LIN {X 0,Y 513.957,Z 334.017,A -85,B 0,C 180,E1 -12997.827,E2 -12997.827} C_VEL
LIN {X 0,Y 513.921,Z 334.019,A -85,B 0,C 180,E1 -13000.86,E2 -13000.86} C_VEL
LIN {X 0,Y 513.953,Z 334.017,A -85,B 0,C 180,E1 -13003.754,E2 -13003.754} C_VEL
LIN {X 0,Y 513.947,Z 334.027,A -85,B 0,C 180,E1 -13007.044,E2 -13007.044} C_VEL
LIN {X 0,Y 513.919,Z 334.024,A -85,B 0,C 180,E1 -13010.164,E2 -13010.164} C_VEL
LIN {X 0,Y 513.918,Z 334.026,A -85,B 0,C 180,E1 -13013.527,E2 -13013.527} C_VEL
LIN {X 0,Y 513.913,Z 334.024,A -85,B 0,C 180,E1 -13016.243,E2 -13016.243} C_VEL
LIN {X 0,Y 513.986,Z 334.221,A -85,B 0,C 180,E1 -13019.321,E2 -13019.321} C_VEL
LIN {X 0,Y 517.909,Z 351.016,A -85,B 0,C 180,E1 -13021.747,E2 -13021.747} C_VEL
LIN {X 0,Y 519.515,Z 360.152,A -85,B 0,C 180,E1 -13023.008,E2 -13023.008} C_VEL
LIN {X 0,Y 518.072,Z 381.283,A -85,B 0,C 180,E1 -13025.646,E2 -13025.646} C_VEL
LIN {X 0,Y 516.469,Z 407.915,A -85,B 0,C 180,E1 -13028.937,E2 -13028.937} C_VEL
LIN {X 0,Y 515.682,Z 421.479,A -85,B 0,C 180,E1 -13030.575,E2 -13030.575} C_VEL
LIN {X 0,Y 517.921,Z 437.713,A -85,B 0,C 180,E1 -13031.06,E2 -13031.06} C_VEL
LIN {X 0,Y 519.767,Z 455.53,A -85,B 0,C 180,E1 -13031.51,E2 -13031.51} C_VEL
LIN {X 0,Y 521.044,Z 469.937,A -85,B 0,C 180,E1 -13031.766,E2 -13031.766} C_VEL
LIN {X 0,Y 519.855,Z 563.729,A -85,B 0,C 180,E1 -13033.083,E2 -13033.083} C_VEL
LIN {X 0,Y 519.209,Z 578.333,A -85,B 0,C 180,E1 -13033.441,E2 -13033.441} C_VEL
LIN {X 0,Y 518.369,Z 591.708,A -85,B 0,C 180,E1 -13033.918,E2 -13033.918} C_VEL
LIN {X 0,Y 517.524,Z 603.945,A -85,B 0,C 180,E1 -13034.496,E2 -13034.496} C_VEL
LIN {X 0,Y 516.53,Z 616.831,A -85,B 0,C 180,E1 -13035.27,E2 -13035.27} C_VEL
LIN {X 0,Y 515.468,Z 629.745,A -85,B 0,C 180,E1 -13036.243,E2 -13036.243} C_VEL
LIN {X 0,Y 514.622,Z 640.615,A -85,B 0,C 180,E1 -13037.222,E2 -13037.222} C_VEL
LIN {X 0,Y 514.134,Z 652.534,A -85,B 0,C 180,E1 -13038.208,E2 -13038.208} C_VEL
LIN {X 0,Y 513.612,Z 663.514,A -85,B 0,C 180,E1 -13039.313,E2 -13039.313} C_VEL
LIN {X 0,Y 513.218,Z 673.738,A -85,B 0,C 180,E1 -13040.574,E2 -13040.574} C_VEL
LIN {X 0,Y 512.862,Z 681.617,A -85,B 0,C 180,E1 -13041.755,E2 -13041.755} C_VEL
LIN {X 0,Y 512.651,Z 688.156,A -85,B 0,C 180,E1 -13042.936,E2 -13042.936} C_VEL
LIN {X 0,Y 512.551,Z 693.504,A -85,B 0,C 180,E1 -13044.117,E2 -13044.117} C_VEL
LIN {X 0,Y 512.438,Z 697.792,A -85,B 0,C 180,E1 -13045.296,E2 -13045.296} C_VEL
LIN {X 0,Y 512.414,Z 700.648,A -85,B 0,C 180,E1 -13046.264,E2 -13046.264} C_VEL
LIN {X 0,Y 512.391,Z 703.639,A -85,B 0,C 180,E1 -13047.649,E2 -13047.649} C_VEL
LIN {X 0,Y 512.384,Z 705.592,A -85,B 0,C 180,E1 -13049.217,E2 -13049.217} C_VEL
LIN {X 0,Y 512.384,Z 706.077,A -85,B 0,C 180,E1 -13050.783,E2 -13050.783} C_VEL
LIN {X 0,Y 512.395,Z 705.11,A -85,B 0,C 180,E1 -13052.35,E2 -13052.35} C_VEL
LIN {X 0,Y 512.438,Z 702.692,A -85,B 0,C 180,E1 -13053.919,E2 -13053.919} C_VEL
LIN {X 0,Y 512.588,Z 698.767,A -85,B 0,C 180,E1 -13055.489,E2 -13055.489} C_VEL
LIN {X 0,Y 512.786,Z 694.711,A -85,B 0,C 180,E1 -13056.667,E2 -13056.667} C_VEL
LIN {X 0,Y 513.044,Z 689.687,A -85,B 0,C 180,E1 -13057.847,E2 -13057.847} C_VEL
LIN {X 0,Y 513.489,Z 682.439,A -85,B 0,C 180,E1 -13059.223,E2 -13059.223} C_VEL
LIN {X 0,Y 514.068,Z 674.823,A -85,B 0,C 180,E1 -13060.401,E2 -13060.401} C_VEL
LIN {X 0,Y 514.707,Z 665.365,A -85,B 0,C 180,E1 -13061.615,E2 -13061.615} C_VEL
LIN {X 0,Y 515.541,Z 654.607,A -85,B 0,C 180,E1 -13062.755,E2 -13062.755} C_VEL
LIN {X 0,Y 516.298,Z 643.373,A -85,B 0,C 180,E1 -13063.734,E2 -13063.734} C_VEL
LIN {X 0,Y 517.195,Z 631.022,A -85,B 0,C 180,E1 -13064.61,E2 -13064.61} C_VEL
LIN {X 0,Y 518.024,Z 617.389,A -85,B 0,C 180,E1 -13065.388,E2 -13065.388} C_VEL
LIN {X 0,Y 518.795,Z 603.147,A -85,B 0,C 180,E1 -13066.018,E2 -13066.018} C_VEL
LIN {X 0,Y 519.42,Z 589.095,A -85,B 0,C 180,E1 -13066.469,E2 -13066.469} C_VEL
LIN {X 0,Y 520.013,Z 571.059,A -85,B 0,C 180,E1 -13066.846,E2 -13066.846} C_VEL
LIN {X 0,Y 522.738,Z 481.781,A -85,B 0,C 180,E1 -13068.556,E2 -13068.556} C_VEL
LIN {X 0,Y 523.003,Z 467.316,A -85,B 0,C 180,E1 -13068.858,E2 -13068.858} C_VEL
LIN {X 0,Y 521.545,Z 448.408,A -85,B 0,C 180,E1 -13069.366,E2 -13069.366} C_VEL
LIN {X 0,Y 519.936,Z 435.629,A -85,B 0,C 180,E1 -13069.758,E2 -13069.758} C_VEL
LIN {X 0,Y 517.568,Z 410.308,A -85,B 0,C 180,E1 -13070.964,E2 -13070.964} C_VEL
LIN {X 0,Y 516.066,Z 396.877,A -85,B 0,C 180,E1 -13071.707,E2 -13071.707} C_VEL
LIN {X 0,Y 517.095,Z 376.419,A -85,B 0,C 180,E1 -13074.19,E2 -13074.19} C_VEL
LIN {X 0,Y 518.269,Z 355.713,A -85,B 0,C 180,E1 -13076.72,E2 -13076.72} C_VEL
LIN {X 0,Y 515.192,Z 339.734,A -85,B 0,C 180,E1 -13078.859,E2 -13078.859} C_VEL
LIN {X 0,Y 514.001,Z 334.02,A -85,B 0,C 180,E1 -13079.659,E2 -13079.659} C_VEL
LIN {X 0,Y 513.908,Z 334.025,A -85,B 0,C 180,E1 -13082.323,E2 -13082.323} C_VEL
LIN {X 0,Y 513.9,Z 334.031,A -85,B 0,C 180,E1 -13085.135,E2 -13085.135} C_VEL
LIN {X 0,Y 513.895,Z 334.026,A -85,B 0,C 180,E1 -13087.832,E2 -13087.832} C_VEL
LIN {X 0,Y 513.915,Z 334.027,A -85,B 0,C 180,E1 -13090.861,E2 -13090.861} C_VEL
LIN {X 0,Y 513.942,Z 334.025,A -85,B 0,C 180,E1 -13094.033,E2 -13094.033} C_VEL
LIN {X 0,Y 513.919,Z 334.025,A -85,B 0,C 180,E1 -13097.041,E2 -13097.041} C_VEL
LIN {X 0,Y 513.918,Z 334.026,A -85,B 0,C 180,E1 -13100.165,E2 -13100.165} C_VEL
LIN {X 0,Y 513.952,Z 334.023,A -85,B 0,C 180,E1 -13103.155,E2 -13103.155} C_VEL
LIN {X 0,Y 513.933,Z 334.027,A -85,B 0,C 180,E1 -13106.24,E2 -13106.24} C_VEL
LIN {X 0,Y 513.966,Z 334.145,A -85,B 0,C 180,E1 -13106.734,E2 -13106.734} C_VEL
LIN {X 0,Y 518.504,Z 346.552,A -85,B 0,C 180,E1 -13108.863,E2 -13108.863} C_VEL
LIN {X 0,Y 522.071,Z 358.438,A -85,B 0,C 180,E1 -13110.702,E2 -13110.702} C_VEL
LIN {X 0,Y 524.202,Z 368.507,A -85,B 0,C 180,E1 -13112.117,E2 -13112.117} C_VEL
LIN {X 0,Y 522.434,Z 393.697,A -85,B 0,C 180,E1 -13115.018,E2 -13115.018} C_VEL
LIN {X 0,Y 520.704,Z 420.277,A -85,B 0,C 180,E1 -13118.029,E2 -13118.029} C_VEL
LIN {X 0,Y 519.609,Z 439.597,A -85,B 0,C 180,E1 -13120.219,E2 -13120.219} C_VEL
LIN {X 0,Y 522.629,Z 456.777,A -85,B 0,C 180,E1 -13120.791,E2 -13120.791} C_VEL
LIN {X 0,Y 523.743,Z 466.69,A -85,B 0,C 180,E1 -13121.071,E2 -13121.071} C_VEL
LIN {X 0,Y 520.924,Z 555.644,A -85,B 0,C 180,E1 -13122.771,E2 -13122.771} C_VEL
LIN {X 0,Y 520.115,Z 582.822,A -85,B 0,C 180,E1 -13123.298,E2 -13123.298} C_VEL
LIN {X 0,Y 519.488,Z 596.312,A -85,B 0,C 180,E1 -13123.703,E2 -13123.703} C_VEL
LIN {X 0,Y 518.707,Z 610.395,A -85,B 0,C 180,E1 -13124.281,E2 -13124.281} C_VEL
LIN {X 0,Y 517.916,Z 624.002,A -85,B 0,C 180,E1 -13125.01,E2 -13125.01} C_VEL
LIN {X 0,Y 517.038,Z 635.75,A -85,B 0,C 180,E1 -13125.786,E2 -13125.786} C_VEL
LIN {X 0,Y 516.1,Z 647.833,A -85,B 0,C 180,E1 -13126.76,E2 -13126.76} C_VEL
LIN {X 0,Y 515.268,Z 658.722,A -85,B 0,C 180,E1 -13127.837,E2 -13127.837} C_VEL
LIN {X 0,Y 514.613,Z 668.576,A -85,B 0,C 180,E1 -13129.015,E2 -13129.015} C_VEL
LIN {X 0,Y 513.925,Z 676.801,A -85,B 0,C 180,E1 -13130.191,E2 -13130.191} C_VEL
LIN {X 0,Y 513.376,Z 684.669,A -85,B 0,C 180,E1 -13131.566,E2 -13131.566} C_VEL
LIN {X 0,Y 512.916,Z 690.978,A -85,B 0,C 180,E1 -13132.94,E2 -13132.94} C_VEL
LIN {X 0,Y 512.627,Z 695.283,A -85,B 0,C 180,E1 -13134.118,E2 -13134.118} C_VEL
LIN {X 0,Y 512.466,Z 698.685,A -85,B 0,C 180,E1 -13135.296,E2 -13135.296} C_VEL
LIN {X 0,Y 512.357,Z 701.825,A -85,B 0,C 180,E1 -13136.865,E2 -13136.865} C_VEL
LIN {X 0,Y 512.309,Z 703.515,A -85,B 0,C 180,E1 -13138.433,E2 -13138.433} C_VEL
LIN {X 0,Y 512.306,Z 703.777,A -85,B 0,C 180,E1 -13140,E2 -13140} C_VEL
LIN {X 0,Y 512.307,Z 702.606,A -85,B 0,C 180,E1 -13141.567,E2 -13141.567} C_VEL
LIN {X 0,Y 512.328,Z 699.97,A -85,B 0,C 180,E1 -13143.135,E2 -13143.135} C_VEL
LIN {X 0,Y 512.418,Z 695.775,A -85,B 0,C 180,E1 -13144.705,E2 -13144.705} C_VEL
LIN {X 0,Y 512.523,Z 691.231,A -85,B 0,C 180,E1 -13145.968,E2 -13145.968} C_VEL
LIN {X 0,Y 512.769,Z 684.336,A -85,B 0,C 180,E1 -13147.457,E2 -13147.457} C_VEL
LIN {X 0,Y 513.092,Z 676.309,A -85,B 0,C 180,E1 -13148.835,E2 -13148.835} C_VEL
LIN {X 0,Y 513.475,Z 667.895,A -85,B 0,C 180,E1 -13150.016,E2 -13150.016} C_VEL
LIN {X 0,Y 514.049,Z 657.233,A -85,B 0,C 180,E1 -13151.251,E2 -13151.251} C_VEL
LIN {X 0,Y 514.52,Z 646.405,A -85,B 0,C 180,E1 -13152.282,E2 -13152.282} C_VEL
LIN {X 0,Y 515.135,Z 633.805,A -85,B 0,C 180,E1 -13153.265,E2 -13153.265} C_VEL
LIN {X 0,Y 515.76,Z 621.419,A -85,B 0,C 180,E1 -13154.05,E2 -13154.05} C_VEL
LIN {X 0,Y 516.376,Z 607.834,A -85,B 0,C 180,E1 -13154.735,E2 -13154.735} C_VEL
LIN {X 0,Y 516.783,Z 593.624,A -85,B 0,C 180,E1 -13155.275,E2 -13155.275} C_VEL
LIN {X 0,Y 517.198,Z 578.976,A -85,B 0,C 180,E1 -13155.665,E2 -13155.665} C_VEL
LIN {X 0,Y 519.097,Z 462.644,A -85,B 0,C 180,E1 -13157.655,E2 -13157.655} C_VEL
LIN {X 0,Y 516.428,Z 439.504,A -85,B 0,C 180,E1 -13158.152,E2 -13158.152} C_VEL
LIN {X 0,Y 517.63,Z 410.077,A -85,B 0,C 180,E1 -13161.43,E2 -13161.43} C_VEL
LIN {X 0,Y 518.796,Z 384.213,A -85,B 0,C 180,E1 -13164.318,E2 -13164.318} C_VEL
LIN {X 0,Y 519.838,Z 360.3,A -85,B 0,C 180,E1 -13167.003,E2 -13167.003} C_VEL
LIN {X 0,Y 515.28,Z 339.725,A -85,B 0,C 180,E1 -13169.543,E2 -13169.543} C_VEL
LIN {X 0,Y 514.013,Z 334.014,A -85,B 0,C 180,E1 -13170.278,E2 -13170.278} C_VEL
LIN {X 0,Y 513.973,Z 334.022,A -85,B 0,C 180,E1 -13173.033,E2 -13173.033} C_VEL
LIN {X 0,Y 513.984,Z 334.015,A -85,B 0,C 180,E1 -13175.874,E2 -13175.874} C_VEL
LIN {X 0,Y 513.947,Z 334.025,A -85,B 0,C 180,E1 -13179.028,E2 -13179.028} C_VEL
LIN {X 0,Y 513.958,Z 334.017,A -85,B 0,C 180,E1 -13181.897,E2 -13181.897} C_VEL
LIN {X 0,Y 513.974,Z 334.021,A -85,B 0,C 180,E1 -13185.126,E2 -13185.126} C_VEL
LIN {X 0,Y 513.959,Z 334.018,A -85,B 0,C 180,E1 -13188.103,E2 -13188.103} C_VEL
LIN {X 0,Y 513.952,Z 334.023,A -85,B 0,C 180,E1 -13190.972,E2 -13190.972} C_VEL
LIN {X 0,Y 513.984,Z 334.016,A -85,B 0,C 180,E1 -13194.127,E2 -13194.127} C_VEL
LIN {X 0,Y 513.962,Z 334.02,A -85,B 0,C 180,E1 -13196.966,E2 -13196.966} C_VEL
LIN {X 0,Y 513.952,Z 334.019,A -85,B 0,C 180,E1 -13199.718,E2 -13199.718} C_VEL
LIN {X 0,Y 513.973,Z 334.024,A -85,B 0,C 180,E1 -13202.396,E2 -13202.396} C_VEL
LIN {X 0,Y 513.933,Z 334.022,A -85,B 0,C 180,E1 -13205.007,E2 -13205.007} C_VEL
LIN {X 0,Y 513.995,Z 334.017,A -85,B 0,C 180,E1 -13207.922,E2 -13207.922} C_VEL
LIN {X 0,Y 513.97,Z 334.017,A -85,B 0,C 180,E1 -13210.909,E2 -13210.909} C_VEL
LIN {X 0,Y 513.973,Z 334.017,A -85,B 0,C 180,E1 -13213.37,E2 -13213.37} C_VEL
LIN {X 0,Y 514.062,Z 334.012,A -85,B 0,C 180,E1 -13215.803,E2 -13215.803} C_VEL
LIN {X 0,Y 514.031,Z 334.01,A -85,B 0,C 180,E1 -13216.922,E2 -13216.922} C_VEL
LIN {X 0,Y 519.318,Z 349.174,A -85,B 0,C 180,E1 -13217.334,E2 -13217.334} C_VEL
LIN {X 0,Y 520.205,Z 352.303,A -85,B 0,C 180,E1 -13217.408,E2 -13217.408} C_VEL
LIN {X 0,Y 519.393,Z 423.895,A -85,B 0,C 180,E1 -13218.392,E2 -13218.392} C_VEL
LIN {X 0,Y 518.705,Z 429.739,A -85,B 0,C 180,E1 -13218.451,E2 -13218.451} C_VEL
LIN {X 0,Y 513.062,Z 448.73,A -85,B 0,C 180,E1 -13218.548,E2 -13218.548} C_VEL
LIN {X 0,Y 512.399,Z 454.555,A -85,B 0,C 180,E1 -13218.625,E2 -13218.625} C_VEL
LIN {X 0,Y 512.285,Z 468.637,A -85,B 0,C 180,E1 -13218.964,E2 -13218.964} C_VEL
LIN {X 0,Y 512.007,Z 482.396,A -85,B 0,C 180,E1 -13219.457,E2 -13219.457} C_VEL
LIN {X 0,Y 511.557,Z 494.768,A -85,B 0,C 180,E1 -13220.046,E2 -13220.046} C_VEL
LIN {X 0,Y 511.014,Z 507.231,A -85,B 0,C 180,E1 -13220.802,E2 -13220.802} C_VEL
LIN {X 0,Y 510.442,Z 519.295,A -85,B 0,C 180,E1 -13221.716,E2 -13221.716} C_VEL
LIN {X 0,Y 509.72,Z 529.971,A -85,B 0,C 180,E1 -13222.697,E2 -13222.697} C_VEL
LIN {X 0,Y 508.908,Z 540.524,A -85,B 0,C 180,E1 -13223.877,E2 -13223.877} C_VEL
LIN {X 0,Y 508.264,Z 549.232,A -85,B 0,C 180,E1 -13225.059,E2 -13225.059} C_VEL
LIN {X 0,Y 507.768,Z 557.559,A -85,B 0,C 180,E1 -13226.441,E2 -13226.441} C_VEL
LIN {X 0,Y 507.204,Z 563.426,A -85,B 0,C 180,E1 -13227.626,E2 -13227.626} C_VEL
LIN {X 0,Y 506.937,Z 568.262,A -85,B 0,C 180,E1 -13228.813,E2 -13228.813} C_VEL
LIN {X 0,Y 506.508,Z 573.278,A -85,B 0,C 180,E1 -13230.396,E2 -13230.396} C_VEL
LIN {X 0,Y 506.46,Z 576.085,A -85,B 0,C 180,E1 -13231.585,E2 -13231.585} C_VEL
LIN {X 0,Y 506.431,Z 578.592,A -85,B 0,C 180,E1 -13233.172,E2 -13233.172} C_VEL
LIN {X 0,Y 506.327,Z 579.803,A -85,B 0,C 180,E1 -13234.761,E2 -13234.761} C_VEL
LIN {X 0,Y 506.447,Z 579.711,A -85,B 0,C 180,E1 -13236.353,E2 -13236.353} C_VEL
LIN {X 0,Y 506.605,Z 578.327,A -85,B 0,C 180,E1 -13237.947,E2 -13237.947} C_VEL
LIN {X 0,Y 506.83,Z 575.611,A -85,B 0,C 180,E1 -13239.546,E2 -13239.546} C_VEL
LIN {X 0,Y 507.376,Z 571.45,A -85,B 0,C 180,E1 -13241.144,E2 -13241.144} C_VEL
LIN {X 0,Y 507.941,Z 565.744,A -85,B 0,C 180,E1 -13242.747,E2 -13242.747} C_VEL
LIN {X 0,Y 508.636,Z 559.28,A -85,B 0,C 180,E1 -13244.149,E2 -13244.149} C_VEL
LIN {X 0,Y 509.328,Z 552.262,A -85,B 0,C 180,E1 -13245.383,E2 -13245.383} C_VEL
LIN {X 0,Y 510.082,Z 544.242,A -85,B 0,C 180,E1 -13246.555,E2 -13246.555} C_VEL
LIN {X 0,Y 510.953,Z 534.314,A -85,B 0,C 180,E1 -13247.759,E2 -13247.759} C_VEL
LIN {X 0,Y 511.859,Z 523.183,A -85,B 0,C 180,E1 -13248.862,E2 -13248.862} C_VEL
LIN {X 0,Y 512.641,Z 512.337,A -85,B 0,C 180,E1 -13249.745,E2 -13249.745} C_VEL
LIN {X 0,Y 513.401,Z 499.868,A -85,B 0,C 180,E1 -13250.568,E2 -13250.568} C_VEL
LIN {X 0,Y 513.807,Z 487.375,A -85,B 0,C 180,E1 -13251.23,E2 -13251.23} C_VEL
LIN {X 0,Y 514.318,Z 473.276,A -85,B 0,C 180,E1 -13251.788,E2 -13251.788} C_VEL
LIN {X 0,Y 514.521,Z 459.871,A -85,B 0,C 180,E1 -13252.165,E2 -13252.165} C_VEL
LIN {X 0,Y 514.657,Z 441.45,A -85,B 0,C 180,E1 -13252.474,E2 -13252.474} C_VEL
LIN {X 0,Y 515.707,Z 356.436,A -85,B 0,C 180,E1 -13253.671,E2 -13253.671} C_VEL
LIN {X 0,Y 506.971,Z 335.261,A -85,B 0,C 180,E1 -13254.373,E2 -13254.373} C_VEL
LIN {X 0,Y 506.897,Z 334.907,A -85,B 0,C 180,E1 -13254.406,E2 -13254.406} C_VEL
LIN {X 0,Y 506.923,Z 334.901,A -85,B 0,C 180,E1 -13257.128,E2 -13257.128} C_VEL
LIN {X 0,Y 506.912,Z 334.902,A -85,B 0,C 180,E1 -13259.831,E2 -13259.831} C_VEL
LIN {X 0,Y 506.853,Z 334.907,A -85,B 0,C 180,E1 -13262.613,E2 -13262.613} C_VEL
LIN {X 0,Y 506.865,Z 334.904,A -85,B 0,C 180,E1 -13265.479,E2 -13265.479} C_VEL
LIN {X 0,Y 506.848,Z 334.909,A -85,B 0,C 180,E1 -13268.027,E2 -13268.027} C_VEL
LIN {X 0,Y 506.871,Z 334.907,A -85,B 0,C 180,E1 -13270.531,E2 -13270.531} C_VEL
LIN {X 0,Y 506.919,Z 334.901,A -85,B 0,C 180,E1 -13273.701,E2 -13273.701} C_VEL
LIN {X 0,Y 506.927,Z 334.895,A -85,B 0,C 180,E1 -13277.082,E2 -13277.082} C_VEL
LIN {X 0,Y 506.885,Z 334.901,A -85,B 0,C 180,E1 -13279.498,E2 -13279.498} C_VEL
LIN {X 0,Y 506.847,Z 334.882,A -85,B 0,C 180,E1 -13282.55,E2 -13282.55} C_VEL
LIN {X 0,Y 506.881,Z 334.891,A -85,B 0,C 180,E1 -13285.488,E2 -13285.488} C_VEL
LIN {X 0,Y 506.885,Z 334.896,A -85,B 0,C 180,E1 -13288.324,E2 -13288.324} C_VEL
LIN {X 0,Y 506.901,Z 334.895,A -85,B 0,C 180,E1 -13291.077,E2 -13291.077} C_VEL
LIN {X 0,Y 506.895,Z 334.895,A -85,B 0,C 180,E1 -13293.922,E2 -13293.922} C_VEL
LIN {X 0,Y 506.879,Z 334.901,A -85,B 0,C 180,E1 -13296.375,E2 -13296.375} C_VEL
LIN {X 0,Y 506.908,Z 334.891,A -85,B 0,C 180,E1 -13298.944,E2 -13298.944} C_VEL
LIN {X 0,Y 506.937,Z 334.903,A -85,B 0,C 180,E1 -13301.265,E2 -13301.265} C_VEL
LIN {X 0,Y 511.935,Z 351.281,A -85,B 0,C 180,E1 -13301.694,E2 -13301.694} C_VEL
LIN {X 0,Y 510.377,Z 454.67,A -85,B 0,C 180,E1 -13303.489,E2 -13303.489} C_VEL
LIN {X 0,Y 510.208,Z 469.999,A -85,B 0,C 180,E1 -13303.93,E2 -13303.93} C_VEL
LIN {X 0,Y 509.876,Z 484.438,A -85,B 0,C 180,E1 -13304.513,E2 -13304.513} C_VEL
LIN {X 0,Y 509.405,Z 498.486,A -85,B 0,C 180,E1 -13305.263,E2 -13305.263} C_VEL
LIN {X 0,Y 508.946,Z 511.86,A -85,B 0,C 180,E1 -13306.165,E2 -13306.165} C_VEL
LIN {X 0,Y 508.389,Z 523.894,A -85,B 0,C 180,E1 -13307.163,E2 -13307.163} C_VEL
LIN {X 0,Y 507.987,Z 534.494,A -85,B 0,C 180,E1 -13308.237,E2 -13308.237} C_VEL
LIN {X 0,Y 507.571,Z 544.547,A -85,B 0,C 180,E1 -13309.464,E2 -13309.464} C_VEL
LIN {X 0,Y 507.126,Z 552.696,A -85,B 0,C 180,E1 -13310.66,E2 -13310.66} C_VEL
LIN {X 0,Y 506.787,Z 560.505,A -85,B 0,C 180,E1 -13312.055,E2 -13312.055} C_VEL
LIN {X 0,Y 506.564,Z 565.914,A -85,B 0,C 180,E1 -13313.25,E2 -13313.25} C_VEL
LIN {X 0,Y 506.416,Z 570.312,A -85,B 0,C 180,E1 -13314.444,E2 -13314.444} C_VEL
LIN {X 0,Y 506.305,Z 574.764,A -85,B 0,C 180,E1 -13316.033,E2 -13316.033} C_VEL
LIN {X 0,Y 506.404,Z 576.408,A -85,B 0,C 180,E1 -13316.828,E2 -13316.828} C_VEL
LIN {X 0,Y 506.258,Z 578.598,A -85,B 0,C 180,E1 -13318.414,E2 -13318.414} C_VEL
LIN {X 0,Y 506.288,Z 579.366,A -85,B 0,C 180,E1 -13320,E2 -13320} C_VEL
LIN {X 0,Y 506.441,Z 578.727,A -85,B 0,C 180,E1 -13321.585,E2 -13321.585} C_VEL
LIN {X 0,Y 506.905,Z 576.644,A -85,B 0,C 180,E1 -13323.168,E2 -13323.168} C_VEL
LIN {X 0,Y 507.463,Z 573.065,A -85,B 0,C 180,E1 -13324.75,E2 -13324.75} C_VEL
LIN {X 0,Y 507.789,Z 567.94,A -85,B 0,C 180,E1 -13326.335,E2 -13326.335} C_VEL
LIN {X 0,Y 508.576,Z 562.047,A -85,B 0,C 180,E1 -13327.697,E2 -13327.697} C_VEL
LIN {X 0,Y 509.344,Z 554.465,A -85,B 0,C 180,E1 -13329.099,E2 -13329.099} C_VEL
LIN {X 0,Y 510.072,Z 546.594,A -85,B 0,C 180,E1 -13330.283,E2 -13330.283} C_VEL
LIN {X 0,Y 510.866,Z 537.044,A -85,B 0,C 180,E1 -13331.467,E2 -13331.467} C_VEL
LIN {X 0,Y 511.625,Z 526.425,A -85,B 0,C 180,E1 -13332.553,E2 -13332.553} C_VEL
LIN {X 0,Y 512.541,Z 514.66,A -85,B 0,C 180,E1 -13333.536,E2 -13333.536} C_VEL
LIN {X 0,Y 513.352,Z 502.575,A -85,B 0,C 180,E1 -13334.358,E2 -13334.358} C_VEL
LIN {X 0,Y 513.923,Z 488.704,A -85,B 0,C 180,E1 -13335.109,E2 -13335.109} C_VEL
LIN {X 0,Y 514.368,Z 474.308,A -85,B 0,C 180,E1 -13335.703,E2 -13335.703} C_VEL
LIN {X 0,Y 514.614,Z 460.05,A -85,B 0,C 180,E1 -13336.126,E2 -13336.126} C_VEL
LIN {X 0,Y 516.808,Z 382.589,A -85,B 0,C 180,E1 -13337.626,E2 -13337.626} C_VEL
LIN {X 0,Y 517.659,Z 357.713,A -85,B 0,C 180,E1 -13338.125,E2 -13338.125} C_VEL
LIN {X 0,Y 511.436,Z 344.312,A -85,B 0,C 180,E1 -13338.832,E2 -13338.832} C_VEL
LIN {X 0,Y 507.821,Z 337.562,A -85,B 0,C 180,E1 -13339.241,E2 -13339.241} C_VEL
LIN {X 0,Y 506.958,Z 334.897,A -85,B 0,C 180,E1 -13339.386,E2 -13339.386} C_VEL
LIN {X 0,Y 506.956,Z 334.899,A -85,B 0,C 180,E1 -13342.222,E2 -13342.222} C_VEL
LIN {X 0,Y 506.886,Z 334.905,A -85,B 0,C 180,E1 -13345.364,E2 -13345.364} C_VEL
LIN {X 0,Y 506.928,Z 334.901,A -85,B 0,C 180,E1 -13348.021,E2 -13348.021} C_VEL
LIN {X 0,Y 506.925,Z 334.897,A -85,B 0,C 180,E1 -13351.053,E2 -13351.053} C_VEL
LIN {X 0,Y 506.909,Z 334.898,A -85,B 0,C 180,E1 -13353.995,E2 -13353.995} C_VEL
LIN {X 0,Y 506.952,Z 334.889,A -85,B 0,C 180,E1 -13356.738,E2 -13356.738} C_VEL
LIN {X 0,Y 506.878,Z 334.901,A -85,B 0,C 180,E1 -13359.469,E2 -13359.469} C_VEL
LIN {X 0,Y 506.924,Z 334.893,A -85,B 0,C 180,E1 -13362.918,E2 -13362.918} C_VEL
LIN {X 0,Y 506.929,Z 334.892,A -85,B 0,C 180,E1 -13366.301,E2 -13366.301} C_VEL
LIN {X 0,Y 506.882,Z 334.901,A -85,B 0,C 180,E1 -13369.497,E2 -13369.497} C_VEL
LIN {X 0,Y 506.848,Z 334.911,A -85,B 0,C 180,E1 -13372.55,E2 -13372.55} C_VEL
LIN {X 0,Y 506.872,Z 334.896,A -85,B 0,C 180,E1 -13375.488,E2 -13375.488} C_VEL
LIN {X 0,Y 506.913,Z 334.902,A -85,B 0,C 180,E1 -13378.949,E2 -13378.949} C_VEL
LIN {X 0,Y 506.894,Z 334.96,A -85,B 0,C 180,E1 -13379.026,E2 -13379.026} C_VEL
LIN {X 0,Y 510.69,Z 350.917,A -85,B 0,C 180,E1 -13381.378,E2 -13381.378} C_VEL
LIN {X 0,Y 512.523,Z 359.992,A -85,B 0,C 180,E1 -13382.664,E2 -13382.664} C_VEL
LIN {X 0,Y 512.344,Z 365.7,A -85,B 0,C 180,E1 -13383.401,E2 -13383.401} C_VEL
LIN {X 0,Y 510.813,Z 387.38,A -85,B 0,C 180,E1 -13386.139,E2 -13386.139} C_VEL
LIN {X 0,Y 509.249,Z 413.325,A -85,B 0,C 180,E1 -13389.385,E2 -13389.385} C_VEL
LIN {X 0,Y 508.854,Z 419.548,A -85,B 0,C 180,E1 -13390.131,E2 -13390.131} C_VEL
LIN {X 0,Y 511.481,Z 437.939,A -85,B 0,C 180,E1 -13390.704,E2 -13390.704} C_VEL
LIN {X 0,Y 513.865,Z 463.849,A -85,B 0,C 180,E1 -13391.397,E2 -13391.397} C_VEL
LIN {X 0,Y 514.331,Z 471.099,A -85,B 0,C 180,E1 -13391.521,E2 -13391.521} C_VEL
LIN {X 0,Y 513.142,Z 562.641,A -85,B 0,C 180,E1 -13392.822,E2 -13392.822} C_VEL
LIN {X 0,Y 512.497,Z 577.276,A -85,B 0,C 180,E1 -13393.183,E2 -13393.183} C_VEL
LIN {X 0,Y 511.527,Z 591.505,A -85,B 0,C 180,E1 -13393.697,E2 -13393.697} C_VEL
LIN {X 0,Y 510.515,Z 605.382,A -85,B 0,C 180,E1 -13394.379,E2 -13394.379} C_VEL
LIN {X 0,Y 509.525,Z 617.843,A -85,B 0,C 180,E1 -13395.165,E2 -13395.165} C_VEL
LIN {X 0,Y 508.45,Z 630.443,A -85,B 0,C 180,E1 -13396.151,E2 -13396.151} C_VEL
LIN {X 0,Y 507.471,Z 642.017,A -85,B 0,C 180,E1 -13397.241,E2 -13397.241} C_VEL
LIN {X 0,Y 507.035,Z 653.715,A -85,B 0,C 180,E1 -13398.243,E2 -13398.243} C_VEL
LIN {X 0,Y 506.531,Z 664.322,A -85,B 0,C 180,E1 -13399.344,E2 -13399.344} C_VEL
LIN {X 0,Y 506.111,Z 674.504,A -85,B 0,C 180,E1 -13400.641,E2 -13400.641} C_VEL
LIN {X 0,Y 505.676,Z 683.413,A -85,B 0,C 180,E1 -13402.038,E2 -13402.038} C_VEL
LIN {X 0,Y 505.522,Z 689.626,A -85,B 0,C 180,E1 -13403.236,E2 -13403.236} C_VEL
LIN {X 0,Y 505.432,Z 694.711,A -85,B 0,C 180,E1 -13404.433,E2 -13404.433} C_VEL
LIN {X 0,Y 505.346,Z 699.905,A -85,B 0,C 180,E1 -13406.026,E2 -13406.026} C_VEL
LIN {X 0,Y 505.293,Z 703.481,A -85,B 0,C 180,E1 -13407.616,E2 -13407.616} C_VEL
LIN {X 0,Y 505.294,Z 705.526,A -85,B 0,C 180,E1 -13409.206,E2 -13409.206} C_VEL
LIN {X 0,Y 505.293,Z 706.076,A -85,B 0,C 180,E1 -13410.794,E2 -13410.794} C_VEL
LIN {X 0,Y 505.298,Z 705.171,A -85,B 0,C 180,E1 -13412.383,E2 -13412.383} C_VEL
LIN {X 0,Y 505.347,Z 702.806,A -85,B 0,C 180,E1 -13413.974,E2 -13413.974} C_VEL
LIN {X 0,Y 505.532,Z 698.941,A -85,B 0,C 180,E1 -13415.566,E2 -13415.566} C_VEL
LIN {X 0,Y 505.734,Z 694.954,A -85,B 0,C 180,E1 -13416.761,E2 -13416.761} C_VEL
LIN {X 0,Y 506.032,Z 689.996,A -85,B 0,C 180,E1 -13417.956,E2 -13417.956} C_VEL
LIN {X 0,Y 506.472,Z 682.805,A -85,B 0,C 180,E1 -13419.352,E2 -13419.352} C_VEL
LIN {X 0,Y 507.238,Z 673.898,A -85,B 0,C 180,E1 -13420.744,E2 -13420.744} C_VEL
LIN {X 0,Y 507.874,Z 664.582,A -85,B 0,C 180,E1 -13421.939,E2 -13421.939} C_VEL
LIN {X 0,Y 508.75,Z 654.273,A -85,B 0,C 180,E1 -13423.029,E2 -13423.029} C_VEL
LIN {X 0,Y 509.505,Z 643.004,A -85,B 0,C 180,E1 -13424.022,E2 -13424.022} C_VEL
LIN {X 0,Y 510.496,Z 630.62,A -85,B 0,C 180,E1 -13424.908,E2 -13424.908} C_VEL
LIN {X 0,Y 511.391,Z 616.918,A -85,B 0,C 180,E1 -13425.695,E2 -13425.695} C_VEL
LIN {X 0,Y 512.208,Z 602.593,A -85,B 0,C 180,E1 -13426.331,E2 -13426.331} C_VEL
LIN {X 0,Y 512.885,Z 588.962,A -85,B 0,C 180,E1 -13426.773,E2 -13426.773} C_VEL
LIN {X 0,Y 513.498,Z 570.893,A -85,B 0,C 180,E1 -13427.16,E2 -13427.16} C_VEL
LIN {X 0,Y 516.394,Z 482.65,A -85,B 0,C 180,E1 -13428.895,E2 -13428.895} C_VEL
LIN {X 0,Y 516.727,Z 468.338,A -85,B 0,C 180,E1 -13429.201,E2 -13429.201} C_VEL
LIN {X 0,Y 515.304,Z 449.521,A -85,B 0,C 180,E1 -13429.723,E2 -13429.723} C_VEL
LIN {X 0,Y 513.603,Z 435.459,A -85,B 0,C 180,E1 -13430.177,E2 -13430.177} C_VEL
LIN {X 0,Y 511.617,Z 413.036,A -85,B 0,C 180,E1 -13431.285,E2 -13431.285} C_VEL
LIN {X 0,Y 509.397,Z 391.831,A -85,B 0,C 180,E1 -13432.511,E2 -13432.511} C_VEL
LIN {X 0,Y 510.896,Z 365.132,A -85,B 0,C 180,E1 -13435.804,E2 -13435.804} C_VEL
LIN {X 0,Y 511.287,Z 356.536,A -85,B 0,C 180,E1 -13436.878,E2 -13436.878} C_VEL
LIN {X 0,Y 507.855,Z 339.069,A -85,B 0,C 180,E1 -13439.257,E2 -13439.257} C_VEL
LIN {X 0,Y 506.949,Z 334.898,A -85,B 0,C 180,E1 -13439.857,E2 -13439.857} C_VEL
LIN {X 0,Y 506.849,Z 334.905,A -85,B 0,C 180,E1 -13442.613,E2 -13442.613} C_VEL
LIN {X 0,Y 506.86,Z 334.904,A -85,B 0,C 180,E1 -13445.479,E2 -13445.479} C_VEL
LIN {X 0,Y 506.837,Z 334.906,A -85,B 0,C 180,E1 -13448.026,E2 -13448.026} C_VEL
LIN {X 0,Y 506.866,Z 334.905,A -85,B 0,C 180,E1 -13450.531,E2 -13450.531} C_VEL
LIN {X 0,Y 506.916,Z 334.901,A -85,B 0,C 180,E1 -13453.7,E2 -13453.7} C_VEL
LIN {X 0,Y 506.916,Z 334.901,A -85,B 0,C 180,E1 -13456.3,E2 -13456.3} C_VEL
LIN {X 0,Y 506.881,Z 334.906,A -85,B 0,C 180,E1 -13459.498,E2 -13459.498} C_VEL
LIN {X 0,Y 506.915,Z 334.901,A -85,B 0,C 180,E1 -13462.556,E2 -13462.556} C_VEL
LIN {X 0,Y 506.894,Z 334.903,A -85,B 0,C 180,E1 -13465.785,E2 -13465.785} C_VEL
LIN {X 0,Y 506.913,Z 335.071,A -85,B 0,C 180,E1 -13466.003,E2 -13466.003} C_VEL
LIN {X 0,Y 511.797,Z 347.857,A -85,B 0,C 180,E1 -13468.319,E2 -13468.319} C_VEL
LIN {X 0,Y 515.702,Z 360.605,A -85,B 0,C 180,E1 -13470.374,E2 -13470.374} C_VEL
LIN {X 0,Y 517.712,Z 369.931,A -85,B 0,C 180,E1 -13471.736,E2 -13471.736} C_VEL
LIN {X 0,Y 517.794,Z 372.577,A -85,B 0,C 180,E1 -13472.072,E2 -13472.072} C_VEL
LIN {X 0,Y 515.83,Z 398.701,A -85,B 0,C 180,E1 -13475.106,E2 -13475.106} C_VEL
LIN {X 0,Y 513.864,Z 427.413,A -85,B 0,C 180,E1 -13478.406,E2 -13478.406} C_VEL
LIN {X 0,Y 513.148,Z 439.953,A -85,B 0,C 180,E1 -13479.822,E2 -13479.822} C_VEL
LIN {X 0,Y 516.088,Z 456.106,A -85,B 0,C 180,E1 -13480.385,E2 -13480.385} C_VEL
LIN {X 0,Y 517.436,Z 467.162,A -85,B 0,C 180,E1 -13480.718,E2 -13480.718} C_VEL
LIN {X 0,Y 514.397,Z 556.843,A -85,B 0,C 180,E1 -13482.476,E2 -13482.476} C_VEL
LIN {X 0,Y 513.578,Z 582.899,A -85,B 0,C 180,E1 -13482.997,E2 -13482.997} C_VEL
LIN {X 0,Y 512.867,Z 597.073,A -85,B 0,C 180,E1 -13483.435,E2 -13483.435} C_VEL
LIN {X 0,Y 512.034,Z 610.919,A -85,B 0,C 180,E1 -13484.02,E2 -13484.02} C_VEL
LIN {X 0,Y 511.258,Z 623.607,A -85,B 0,C 180,E1 -13484.708,E2 -13484.708} C_VEL
LIN {X 0,Y 510.381,Z 635.387,A -85,B 0,C 180,E1 -13485.495,E2 -13485.495} C_VEL
LIN {X 0,Y 509.338,Z 647.519,A -85,B 0,C 180,E1 -13486.48,E2 -13486.48} C_VEL
LIN {X 0,Y 508.533,Z 657.571,A -85,B 0,C 180,E1 -13487.471,E2 -13487.471} C_VEL
LIN {X 0,Y 507.844,Z 666.396,A -85,B 0,C 180,E1 -13488.503,E2 -13488.503} C_VEL
LIN {X 0,Y 507.104,Z 676.004,A -85,B 0,C 180,E1 -13489.857,E2 -13489.857} C_VEL
LIN {X 0,Y 506.377,Z 684.02,A -85,B 0,C 180,E1 -13491.248,E2 -13491.248} C_VEL
LIN {X 0,Y 505.962,Z 689.646,A -85,B 0,C 180,E1 -13492.443,E2 -13492.443} C_VEL
LIN {X 0,Y 505.586,Z 695.523,A -85,B 0,C 180,E1 -13494.036,E2 -13494.036} C_VEL
LIN {X 0,Y 505.401,Z 698.862,A -85,B 0,C 180,E1 -13495.23,E2 -13495.23} C_VEL
LIN {X 0,Y 505.275,Z 701.946,A -85,B 0,C 180,E1 -13496.821,E2 -13496.821} C_VEL
LIN {X 0,Y 505.226,Z 703.578,A -85,B 0,C 180,E1 -13498.411,E2 -13498.411} C_VEL
LIN {X 0,Y 505.217,Z 703.778,A -85,B 0,C 180,E1 -13500,E2 -13500} C_VEL
LIN {X 0,Y 505.224,Z 702.539,A -85,B 0,C 180,E1 -13501.589,E2 -13501.589} C_VEL
LIN {X 0,Y 505.229,Z 699.804,A -85,B 0,C 180,E1 -13503.179,E2 -13503.179} C_VEL
LIN {X 0,Y 505.338,Z 695.531,A -85,B 0,C 180,E1 -13504.771,E2 -13504.771} C_VEL
LIN {X 0,Y 505.429,Z 691.229,A -85,B 0,C 180,E1 -13505.973,E2 -13505.973} C_VEL
LIN {X 0,Y 505.653,Z 684.938,A -85,B 0,C 180,E1 -13507.362,E2 -13507.362} C_VEL
LIN {X 0,Y 505.977,Z 677.023,A -85,B 0,C 180,E1 -13508.759,E2 -13508.759} C_VEL
LIN {X 0,Y 506.354,Z 668.736,A -85,B 0,C 180,E1 -13509.958,E2 -13509.958} C_VEL
LIN {X 0,Y 506.893,Z 658.755,A -85,B 0,C 180,E1 -13511.155,E2 -13511.155} C_VEL
LIN {X 0,Y 507.427,Z 647.67,A -85,B 0,C 180,E1 -13512.254,E2 -13512.254} C_VEL
LIN {X 0,Y 508.005,Z 635.308,A -85,B 0,C 180,E1 -13513.252,E2 -13513.252} C_VEL
LIN {X 0,Y 508.735,Z 621.558,A -85,B 0,C 180,E1 -13514.146,E2 -13514.146} C_VEL
LIN {X 0,Y 509.353,Z 608.013,A -85,B 0,C 180,E1 -13514.84,E2 -13514.84} C_VEL
LIN {X 0,Y 509.775,Z 593.903,A -85,B 0,C 180,E1 -13515.389,E2 -13515.389} C_VEL
LIN {X 0,Y 510.198,Z 579.425,A -85,B 0,C 180,E1 -13515.784,E2 -13515.784} C_VEL
LIN {X 0,Y 512.213,Z 463.531,A -85,B 0,C 180,E1 -13517.817,E2 -13517.817} C_VEL
LIN {X 0,Y 509.475,Z 439.585,A -85,B 0,C 180,E1 -13518.331,E2 -13518.331} C_VEL
LIN {X 0,Y 510.771,Z 409.281,A -85,B 0,C 180,E1 -13521.732,E2 -13521.732} C_VEL
LIN {X 0,Y 511.998,Z 383.288,A -85,B 0,C 180,E1 -13524.662,E2 -13524.662} C_VEL
LIN {X 0,Y 512.937,Z 361.83,A -85,B 0,C 180,E1 -13527.09,E2 -13527.09} C_VEL
LIN {X 0,Y 508.54,Z 341.92,A -85,B 0,C 180,E1 -13529.572,E2 -13529.572} C_VEL
LIN {X 0,Y 506.941,Z 334.895,A -85,B 0,C 180,E1 -13530.459,E2 -13530.459} C_VEL
LIN {X 0,Y 506.91,Z 334.9,A -85,B 0,C 180,E1 -13533.554,E2 -13533.554} C_VEL
LIN {X 0,Y 506.952,Z 334.892,A -85,B 0,C 180,E1 -13536.739,E2 -13536.739} C_VEL
LIN {X 0,Y 506.923,Z 334.897,A -85,B 0,C 180,E1 -13539.466,E2 -13539.466} C_VEL
LIN {X 0,Y 506.915,Z 334.898,A -85,B 0,C 180,E1 -13542.616,E2 -13542.616} C_VEL
LIN {X 0,Y 506.931,Z 334.898,A -85,B 0,C 180,E1 -13545.196,E2 -13545.196} C_VEL
LIN {X 0,Y 506.911,Z 334.896,A -85,B 0,C 180,E1 -13548.26,E2 -13548.26} C_VEL
LIN {X 0,Y 506.929,Z 334.9,A -85,B 0,C 180,E1 -13550.695,E2 -13550.695} C_VEL
LIN {X 0,Y 506.962,Z 334.889,A -85,B 0,C 180,E1 -13553.551,E2 -13553.551} C_VEL
LIN {X 0,Y 506.918,Z 334.901,A -85,B 0,C 180,E1 -13556.447,E2 -13556.447} C_VEL
LIN {X 0,Y 506.904,Z 334.897,A -85,B 0,C 180,E1 -13559.252,E2 -13559.252} C_VEL
LIN {X 0,Y 506.941,Z 334.896,A -85,B 0,C 180,E1 -13562.165,E2 -13562.165} C_VEL
LIN {X 0,Y 506.913,Z 334.895,A -85,B 0,C 180,E1 -13565.51,E2 -13565.51} C_VEL
LIN {X 0,Y 506.953,Z 334.897,A -85,B 0,C 180,E1 -13568.096,E2 -13568.096} C_VEL
LIN {X 0,Y 506.933,Z 334.895,A -85,B 0,C 180,E1 -13570.633,E2 -13570.633} C_VEL
LIN {X 0,Y 506.939,Z 334.892,A -85,B 0,C 180,E1 -13573.133,E2 -13573.133} C_VEL
LIN {X 0,Y 507.021,Z 334.889,A -85,B 0,C 180,E1 -13575.601,E2 -13575.601} C_VEL
LIN {X 0,Y 506.988,Z 334.887,A -85,B 0,C 180,E1 -13576.709,E2 -13576.709} C_VEL
LIN {X 0,Y 513.395,Z 353.613,A -85,B 0,C 180,E1 -13577.2,E2 -13577.2} C_VEL
LIN {X 0,Y 512.451,Z 451.149,A -85,B 0,C 180,E1 -13578.569,E2 -13578.569} C_VEL
LIN {X 0,Y 512.399,Z 454.555,A -85,B 0,C 180,E1 -13578.625,E2 -13578.625} C_VEL
LIN {X 0,Y 511.701,Z 460.38,A -85,B 0,C 180,E1 -13578.718,E2 -13578.718} C_VEL
LIN {X 0,Y 508.767,Z 469.777,A -85,B 0,C 180,E1 -13578.875,E2 -13578.875} C_VEL
LIN {X 0,Y 505.821,Z 478.992,A -85,B 0,C 180,E1 -13579.112,E2 -13579.112} C_VEL
LIN {X 0,Y 505.101,Z 484.521,A -85,B 0,C 180,E1 -13579.327,E2 -13579.327} C_VEL
LIN {X 0,Y 504.604,Z 498.044,A -85,B 0,C 180,E1 -13580.008,E2 -13580.008} C_VEL
LIN {X 0,Y 504.078,Z 510.232,A -85,B 0,C 180,E1 -13580.791,E2 -13580.791} C_VEL
LIN {X 0,Y 503.439,Z 521.728,A -85,B 0,C 180,E1 -13581.7,E2 -13581.7} C_VEL
LIN {X 0,Y 502.608,Z 533.081,A -85,B 0,C 180,E1 -13582.795,E2 -13582.795} C_VEL
LIN {X 0,Y 501.796,Z 543.243,A -85,B 0,C 180,E1 -13583.991,E2 -13583.991} C_VEL
LIN {X 0,Y 501.181,Z 551.619,A -85,B 0,C 180,E1 -13585.19,E2 -13585.19} C_VEL
LIN {X 0,Y 500.606,Z 559.642,A -85,B 0,C 180,E1 -13586.591,E2 -13586.591} C_VEL
LIN {X 0,Y 500.146,Z 566.107,A -85,B 0,C 180,E1 -13587.994,E2 -13587.994} C_VEL
LIN {X 0,Y 499.62,Z 571.87,A -85,B 0,C 180,E1 -13589.598,E2 -13589.598} C_VEL
LIN {X 0,Y 499.442,Z 575.197,A -85,B 0,C 180,E1 -13590.804,E2 -13590.804} C_VEL
LIN {X 0,Y 499.372,Z 578.339,A -85,B 0,C 180,E1 -13592.412,E2 -13592.412} C_VEL
LIN {X 0,Y 499.25,Z 580.16,A -85,B 0,C 180,E1 -13594.023,E2 -13594.023} C_VEL
LIN {X 0,Y 499.362,Z 580.674,A -85,B 0,C 180,E1 -13595.635,E2 -13595.635} C_VEL
LIN {X 0,Y 499.474,Z 579.908,A -85,B 0,C 180,E1 -13597.251,E2 -13597.251} C_VEL
LIN {X 0,Y 499.682,Z 577.83,A -85,B 0,C 180,E1 -13598.87,E2 -13598.87} C_VEL
LIN {X 0,Y 500.168,Z 574.36,A -85,B 0,C 180,E1 -13600.49,E2 -13600.49} C_VEL
LIN {X 0,Y 500.654,Z 569.416,A -85,B 0,C 180,E1 -13602.114,E2 -13602.114} C_VEL
LIN {X 0,Y 501.208,Z 564.595,A -85,B 0,C 180,E1 -13603.332,E2 -13603.332} C_VEL
LIN {X 0,Y 501.956,Z 557.645,A -85,B 0,C 180,E1 -13604.754,E2 -13604.754} C_VEL
LIN {X 0,Y 502.86,Z 549.005,A -85,B 0,C 180,E1 -13606.176,E2 -13606.176} C_VEL
LIN {X 0,Y 503.724,Z 539.924,A -85,B 0,C 180,E1 -13607.396,E2 -13607.396} C_VEL
LIN {X 0,Y 504.553,Z 529.858,A -85,B 0,C 180,E1 -13608.516,E2 -13608.516} C_VEL
LIN {X 0,Y 505.391,Z 518.743,A -85,B 0,C 180,E1 -13609.533,E2 -13609.533} C_VEL
LIN {X 0,Y 506.335,Z 506.367,A -85,B 0,C 180,E1 -13610.445,E2 -13610.445} C_VEL
LIN {X 0,Y 506.987,Z 494.394,A -85,B 0,C 180,E1 -13611.158,E2 -13611.158} C_VEL
LIN {X 0,Y 507.374,Z 482.5,A -85,B 0,C 180,E1 -13611.725,E2 -13611.725} C_VEL
LIN {X 0,Y 507.784,Z 468.407,A -85,B 0,C 180,E1 -13612.22,E2 -13612.22} C_VEL
LIN {X 0,Y 507.929,Z 455.496,A -85,B 0,C 180,E1 -13612.531,E2 -13612.531} C_VEL
LIN {X 0,Y 509.06,Z 358.122,A -85,B 0,C 180,E1 -13613.938,E2 -13613.938} C_VEL
LIN {X 0,Y 499.932,Z 336.2,A -85,B 0,C 180,E1 -13614.684,E2 -13614.684} C_VEL
LIN {X 0,Y 499.857,Z 335.786,A -85,B 0,C 180,E1 -13614.719,E2 -13614.719} C_VEL
LIN {X 0,Y 499.847,Z 335.782,A -85,B 0,C 180,E1 -13617.545,E2 -13617.545} C_VEL
LIN {X 0,Y 499.848,Z 335.782,A -85,B 0,C 180,E1 -13620.297,E2 -13620.297} C_VEL
LIN {X 0,Y 499.801,Z 335.783,A -85,B 0,C 180,E1 -13623.132,E2 -13623.132} C_VEL
LIN {X 0,Y 499.813,Z 335.785,A -85,B 0,C 180,E1 -13626.058,E2 -13626.058} C_VEL
LIN {X 0,Y 499.821,Z 335.781,A -85,B 0,C 180,E1 -13629.097,E2 -13629.097} C_VEL
LIN {X 0,Y 499.821,Z 335.785,A -85,B 0,C 180,E1 -13632.274,E2 -13632.274} C_VEL
LIN {X 0,Y 499.855,Z 335.776,A -85,B 0,C 180,E1 -13634.479,E2 -13634.479} C_VEL
LIN {X 0,Y 499.882,Z 335.773,A -85,B 0,C 180,E1 -13636.772,E2 -13636.772} C_VEL
LIN {X 0,Y 499.828,Z 335.785,A -85,B 0,C 180,E1 -13639.862,E2 -13639.862} C_VEL
LIN {X 0,Y 499.833,Z 335.754,A -85,B 0,C 180,E1 -13643.014,E2 -13643.014} C_VEL
LIN {X 0,Y 499.842,Z 335.774,A -85,B 0,C 180,E1 -13645.907,E2 -13645.907} C_VEL
LIN {X 0,Y 499.84,Z 335.771,A -85,B 0,C 180,E1 -13648.768,E2 -13648.768} C_VEL
LIN {X 0,Y 499.84,Z 335.78,A -85,B 0,C 180,E1 -13651.546,E2 -13651.546} C_VEL
LIN {X 0,Y 499.832,Z 335.774,A -85,B 0,C 180,E1 -13654.251,E2 -13654.251} C_VEL
LIN {X 0,Y 499.818,Z 335.78,A -85,B 0,C 180,E1 -13656.896,E2 -13656.896} C_VEL
LIN {X 0,Y 499.88,Z 335.779,A -85,B 0,C 180,E1 -13659.856,E2 -13659.856} C_VEL
LIN {X 0,Y 499.892,Z 335.778,A -85,B 0,C 180,E1 -13661.093,E2 -13661.093} C_VEL
LIN {X 0,Y 505.041,Z 352.762,A -85,B 0,C 180,E1 -13661.549,E2 -13661.549} C_VEL
LIN {X 0,Y 503.412,Z 454.652,A -85,B 0,C 180,E1 -13663.349,E2 -13663.349} C_VEL
LIN {X 0,Y 503.228,Z 469.84,A -85,B 0,C 180,E1 -13663.784,E2 -13663.784} C_VEL
LIN {X 0,Y 502.874,Z 484.031,A -85,B 0,C 180,E1 -13664.354,E2 -13664.354} C_VEL
LIN {X 0,Y 502.483,Z 497.405,A -85,B 0,C 180,E1 -13665.055,E2 -13665.055} C_VEL
LIN {X 0,Y 501.992,Z 511.103,A -85,B 0,C 180,E1 -13665.969,E2 -13665.969} C_VEL
LIN {X 0,Y 501.416,Z 523.422,A -85,B 0,C 180,E1 -13666.982,E2 -13666.982} C_VEL
LIN {X 0,Y 501.026,Z 533.965,A -85,B 0,C 180,E1 -13668.034,E2 -13668.034} C_VEL
LIN {X 0,Y 500.578,Z 544.512,A -85,B 0,C 180,E1 -13669.315,E2 -13669.315} C_VEL
LIN {X 0,Y 500.099,Z 552.803,A -85,B 0,C 180,E1 -13670.527,E2 -13670.527} C_VEL
LIN {X 0,Y 499.741,Z 560.74,A -85,B 0,C 180,E1 -13671.943,E2 -13671.943} C_VEL
LIN {X 0,Y 499.505,Z 566.266,A -85,B 0,C 180,E1 -13673.154,E2 -13673.154} C_VEL
LIN {X 0,Y 499.369,Z 570.772,A -85,B 0,C 180,E1 -13674.365,E2 -13674.365} C_VEL
LIN {X 0,Y 499.245,Z 575.329,A -85,B 0,C 180,E1 -13675.977,E2 -13675.977} C_VEL
LIN {X 0,Y 499.348,Z 577.027,A -85,B 0,C 180,E1 -13676.783,E2 -13676.783} C_VEL
LIN {X 0,Y 499.212,Z 579.352,A -85,B 0,C 180,E1 -13678.392,E2 -13678.392} C_VEL
LIN {X 0,Y 499.264,Z 580.211,A -85,B 0,C 180,E1 -13680,E2 -13680} C_VEL
LIN {X 0,Y 499.422,Z 579.661,A -85,B 0,C 180,E1 -13681.607,E2 -13681.607} C_VEL
LIN {X 0,Y 499.899,Z 577.669,A -85,B 0,C 180,E1 -13683.213,E2 -13683.213} C_VEL
LIN {X 0,Y 500.48,Z 574.21,A -85,B 0,C 180,E1 -13684.817,E2 -13684.817} C_VEL
LIN {X 0,Y 500.847,Z 569.171,A -85,B 0,C 180,E1 -13686.424,E2 -13686.424} C_VEL
LIN {X 0,Y 501.675,Z 563.379,A -85,B 0,C 180,E1 -13687.804,E2 -13687.804} C_VEL
LIN {X 0,Y 502.501,Z 555.901,A -85,B 0,C 180,E1 -13689.224,E2 -13689.224} C_VEL
LIN {X 0,Y 503.248,Z 548.131,A -85,B 0,C 180,E1 -13690.424,E2 -13690.424} C_VEL
LIN {X 0,Y 504.093,Z 538.781,A -85,B 0,C 180,E1 -13691.623,E2 -13691.623} C_VEL
LIN {X 0,Y 504.869,Z 528.363,A -85,B 0,C 180,E1 -13692.723,E2 -13692.723} C_VEL
LIN {X 0,Y 505.866,Z 516.479,A -85,B 0,C 180,E1 -13693.741,E2 -13693.741} C_VEL
LIN {X 0,Y 506.839,Z 503.062,A -85,B 0,C 180,E1 -13694.671,E2 -13694.671} C_VEL
LIN {X 0,Y 507.423,Z 489.589,A -85,B 0,C 180,E1 -13695.41,E2 -13695.41} C_VEL
LIN {X 0,Y 507.874,Z 475.274,A -85,B 0,C 180,E1 -13696.012,E2 -13696.012} C_VEL
LIN {X 0,Y 508.164,Z 461.03,A -85,B 0,C 180,E1 -13696.439,E2 -13696.439} C_VEL
LIN {X 0,Y 510.393,Z 386.589,A -85,B 0,C 180,E1 -13697.923,E2 -13697.923} C_VEL
LIN {X 0,Y 511.382,Z 359.742,A -85,B 0,C 180,E1 -13698.474,E2 -13698.474} C_VEL
LIN {X 0,Y 504.839,Z 345.809,A -85,B 0,C 180,E1 -13699.248,E2 -13699.248} C_VEL
LIN {X 0,Y 500.19,Z 336.949,A -85,B 0,C 180,E1 -13699.808,E2 -13699.808} C_VEL
LIN {X 0,Y 499.928,Z 335.772,A -85,B 0,C 180,E1 -13699.863,E2 -13699.863} C_VEL
LIN {X 0,Y 499.908,Z 335.776,A -85,B 0,C 180,E1 -13702.367,E2 -13702.367} C_VEL
LIN {X 0,Y 499.851,Z 335.78,A -85,B 0,C 180,E1 -13704.859,E2 -13704.859} C_VEL
LIN {X 0,Y 499.883,Z 335.777,A -85,B 0,C 180,E1 -13707.542,E2 -13707.542} C_VEL
LIN {X 0,Y 499.853,Z 335.778,A -85,B 0,C 180,E1 -13710.296,E2 -13710.296} C_VEL
LIN {X 0,Y 499.87,Z 335.777,A -85,B 0,C 180,E1 -13713.126,E2 -13713.126} C_VEL
LIN {X 0,Y 499.908,Z 335.767,A -85,B 0,C 180,E1 -13716.049,E2 -13716.049} C_VEL
LIN {X 0,Y 499.841,Z 335.773,A -85,B 0,C 180,E1 -13719.094,E2 -13719.094} C_VEL
LIN {X 0,Y 499.843,Z 335.772,A -85,B 0,C 180,E1 -13722.271,E2 -13722.271} C_VEL
LIN {X 0,Y 499.855,Z 335.773,A -85,B 0,C 180,E1 -13724.479,E2 -13724.479} C_VEL
LIN {X 0,Y 499.879,Z 335.775,A -85,B 0,C 180,E1 -13726.772,E2 -13726.772} C_VEL
LIN {X 0,Y 499.825,Z 335.779,A -85,B 0,C 180,E1 -13729.861,E2 -13729.861} C_VEL
LIN {X 0,Y 499.831,Z 335.781,A -85,B 0,C 180,E1 -13733.013,E2 -13733.013} C_VEL
LIN {X 0,Y 499.829,Z 335.775,A -85,B 0,C 180,E1 -13735.906,E2 -13735.906} C_VEL
LIN {X 0,Y 499.855,Z 335.785,A -85,B 0,C 180,E1 -13738.736,E2 -13738.736} C_VEL
LIN {X 0,Y 503.73,Z 351.976,A -85,B 0,C 180,E1 -13741.166,E2 -13741.166} C_VEL
LIN {X 0,Y 505.722,Z 362.116,A -85,B 0,C 180,E1 -13742.623,E2 -13742.623} C_VEL
LIN {X 0,Y 504.737,Z 376.819,A -85,B 0,C 180,E1 -13744.519,E2 -13744.519} C_VEL
LIN {X 0,Y 503.028,Z 401.784,A -85,B 0,C 180,E1 -13747.701,E2 -13747.701} C_VEL
LIN {X 0,Y 502.079,Z 417.124,A -85,B 0,C 180,E1 -13749.641,E2 -13749.641} C_VEL
LIN {X 0,Y 505.13,Z 438.54,A -85,B 0,C 180,E1 -13750.343,E2 -13750.343} C_VEL
LIN {X 0,Y 507.578,Z 466.931,A -85,B 0,C 180,E1 -13751.131,E2 -13751.131} C_VEL
LIN {X 0,Y 507.605,Z 473.425,A -85,B 0,C 180,E1 -13751.277,E2 -13751.277} C_VEL
LIN {X 0,Y 506.418,Z 562.363,A -85,B 0,C 180,E1 -13752.57,E2 -13752.57} C_VEL
LIN {X 0,Y 505.766,Z 576.825,A -85,B 0,C 180,E1 -13752.936,E2 -13752.936} C_VEL
LIN {X 0,Y 504.805,Z 590.195,A -85,B 0,C 180,E1 -13753.422,E2 -13753.422} C_VEL
LIN {X 0,Y 503.854,Z 603.303,A -85,B 0,C 180,E1 -13754.064,E2 -13754.064} C_VEL
LIN {X 0,Y 502.773,Z 616.008,A -85,B 0,C 180,E1 -13754.857,E2 -13754.857} C_VEL
LIN {X 0,Y 501.74,Z 627.612,A -85,B 0,C 180,E1 -13755.756,E2 -13755.756} C_VEL
LIN {X 0,Y 500.833,Z 637.31,A -85,B 0,C 180,E1 -13756.658,E2 -13756.658} C_VEL
LIN {X 0,Y 500.418,Z 642.085,A -85,B 0,C 180,E1 -13757.161,E2 -13757.161} C_VEL
LIN {X 0,Y 499.982,Z 653.771,A -85,B 0,C 180,E1 -13758.177,E2 -13758.177} C_VEL
LIN {X 0,Y 499.436,Z 664.624,A -85,B 0,C 180,E1 -13759.324,E2 -13759.324} C_VEL
LIN {X 0,Y 499.064,Z 673.846,A -85,B 0,C 180,E1 -13760.508,E2 -13760.508} C_VEL
LIN {X 0,Y 498.69,Z 681.715,A -85,B 0,C 180,E1 -13761.722,E2 -13761.722} C_VEL
LIN {X 0,Y 498.447,Z 689.186,A -85,B 0,C 180,E1 -13763.14,E2 -13763.14} C_VEL
LIN {X 0,Y 498.357,Z 694.365,A -85,B 0,C 180,E1 -13764.354,E2 -13764.354} C_VEL
LIN {X 0,Y 498.246,Z 699.643,A -85,B 0,C 180,E1 -13765.969,E2 -13765.969} C_VEL
LIN {X 0,Y 498.199,Z 703.302,A -85,B 0,C 180,E1 -13767.582,E2 -13767.582} C_VEL
LIN {X 0,Y 498.206,Z 705.443,A -85,B 0,C 180,E1 -13769.194,E2 -13769.194} C_VEL
LIN {X 0,Y 498.205,Z 706.076,A -85,B 0,C 180,E1 -13770.805,E2 -13770.805} C_VEL
LIN {X 0,Y 498.204,Z 705.235,A -85,B 0,C 180,E1 -13772.417,E2 -13772.417} C_VEL
LIN {X 0,Y 498.253,Z 702.939,A -85,B 0,C 180,E1 -13774.031,E2 -13774.031} C_VEL
LIN {X 0,Y 498.468,Z 699.133,A -85,B 0,C 180,E1 -13775.645,E2 -13775.645} C_VEL
LIN {X 0,Y 498.767,Z 693.722,A -85,B 0,C 180,E1 -13777.261,E2 -13777.261} C_VEL
LIN {X 0,Y 499.181,Z 687.494,A -85,B 0,C 180,E1 -13778.676,E2 -13778.676} C_VEL
LIN {X 0,Y 499.85,Z 679.672,A -85,B 0,C 180,E1 -13780.088,E2 -13780.088} C_VEL
LIN {X 0,Y 500.535,Z 670.712,A -85,B 0,C 180,E1 -13781.407,E2 -13781.407} C_VEL
LIN {X 0,Y 501.29,Z 661.701,A -85,B 0,C 180,E1 -13782.508,E2 -13782.508} C_VEL
LIN {X 0,Y 502.355,Z 649.75,A -85,B 0,C 180,E1 -13783.712,E2 -13783.712} C_VEL
LIN {X 0,Y 503.144,Z 638.875,A -85,B 0,C 180,E1 -13784.615,E2 -13784.615} C_VEL
LIN {X 0,Y 504.22,Z 625.549,A -85,B 0,C 180,E1 -13785.51,E2 -13785.51} C_VEL
LIN {X 0,Y 505.086,Z 611.51,A -85,B 0,C 180,E1 -13786.258,E2 -13786.258} C_VEL
LIN {X 0,Y 505.932,Z 596.754,A -85,B 0,C 180,E1 -13786.85,E2 -13786.85} C_VEL
LIN {X 0,Y 506.653,Z 582.06,A -85,B 0,C 180,E1 -13787.26,E2 -13787.26} C_VEL
LIN {X 0,Y 510.013,Z 485.396,A -85,B 0,C 180,E1 -13789.213,E2 -13789.213} C_VEL
LIN {X 0,Y 510.465,Z 469.191,A -85,B 0,C 180,E1 -13789.564,E2 -13789.564} C_VEL
LIN {X 0,Y 509.094,Z 449.884,A -85,B 0,C 180,E1 -13790.119,E2 -13790.119} C_VEL
LIN {X 0,Y 507.296,Z 435.248,A -85,B 0,C 180,E1 -13790.615,E2 -13790.615} C_VEL
LIN {X 0,Y 505.558,Z 414.09,A -85,B 0,C 180,E1 -13791.706,E2 -13791.706} C_VEL
LIN {X 0,Y 503.23,Z 391.595,A -85,B 0,C 180,E1 -13793.068,E2 -13793.068} C_VEL
LIN {X 0,Y 502.798,Z 385.769,A -85,B 0,C 180,E1 -13793.466,E2 -13793.466} C_VEL
LIN {X 0,Y 504.386,Z 358.963,A -85,B 0,C 180,E1 -13796.829,E2 -13796.829} C_VEL
LIN {X 0,Y 502.877,Z 350.056,A -85,B 0,C 180,E1 -13798.04,E2 -13798.04} C_VEL
LIN {X 0,Y 499.903,Z 335.774,A -85,B 0,C 180,E1 -13800.053,E2 -13800.053} C_VEL
LIN {X 0,Y 499.797,Z 335.788,A -85,B 0,C 180,E1 -13803.132,E2 -13803.132} C_VEL
LIN {X 0,Y 499.807,Z 335.781,A -85,B 0,C 180,E1 -13806.058,E2 -13806.058} C_VEL
LIN {X 0,Y 499.814,Z 335.781,A -85,B 0,C 180,E1 -13809.097,E2 -13809.097} C_VEL
LIN {X 0,Y 499.817,Z 335.784,A -85,B 0,C 180,E1 -13812.274,E2 -13812.274} C_VEL
LIN {X 0,Y 499.851,Z 335.782,A -85,B 0,C 180,E1 -13814.479,E2 -13814.479} C_VEL
LIN {X 0,Y 499.864,Z 335.776,A -85,B 0,C 180,E1 -13816.774,E2 -13816.774} C_VEL
LIN {X 0,Y 499.824,Z 335.783,A -85,B 0,C 180,E1 -13819.862,E2 -13819.862} C_VEL
LIN {X 0,Y 499.886,Z 335.776,A -85,B 0,C 180,E1 -13823.005,E2 -13823.005} C_VEL
LIN {X 0,Y 499.863,Z 335.863,A -85,B 0,C 180,E1 -13825.161,E2 -13825.161} C_VEL
LIN {X 0,Y 504.491,Z 347.767,A -85,B 0,C 180,E1 -13827.471,E2 -13827.471} C_VEL
LIN {X 0,Y 507.542,Z 356.71,A -85,B 0,C 180,E1 -13829.032,E2 -13829.032} C_VEL
LIN {X 0,Y 510.261,Z 366.613,A -85,B 0,C 180,E1 -13830.611,E2 -13830.611} C_VEL
LIN {X 0,Y 511.574,Z 373.415,A -85,B 0,C 180,E1 -13831.612,E2 -13831.612} C_VEL
LIN {X 0,Y 509.942,Z 394.695,A -85,B 0,C 180,E1 -13834.144,E2 -13834.144} C_VEL
LIN {X 0,Y 507.68,Z 424.167,A -85,B 0,C 180,E1 -13837.578,E2 -13837.578} C_VEL
LIN {X 0,Y 506.703,Z 439.97,A -85,B 0,C 180,E1 -13839.389,E2 -13839.389} C_VEL
LIN {X 0,Y 509.944,Z 457.659,A -85,B 0,C 180,E1 -13840.033,E2 -13840.033} C_VEL
LIN {X 0,Y 511.154,Z 467.648,A -85,B 0,C 180,E1 -13840.347,E2 -13840.347} C_VEL
LIN {X 0,Y 508.114,Z 552.815,A -85,B 0,C 180,E1 -13842.067,E2 -13842.067} C_VEL
LIN {X 0,Y 507.065,Z 582.666,A -85,B 0,C 180,E1 -13842.672,E2 -13842.672} C_VEL
LIN {X 0,Y 506.293,Z 596.714,A -85,B 0,C 180,E1 -13843.11,E2 -13843.11} C_VEL
LIN {X 0,Y 505.426,Z 610.632,A -85,B 0,C 180,E1 -13843.702,E2 -13843.702} C_VEL
LIN {X 0,Y 504.621,Z 623.319,A -85,B 0,C 180,E1 -13844.399,E2 -13844.399} C_VEL
LIN {X 0,Y 503.677,Z 635.115,A -85,B 0,C 180,E1 -13845.195,E2 -13845.195} C_VEL
LIN {X 0,Y 502.623,Z 647.276,A -85,B 0,C 180,E1 -13846.193,E2 -13846.193} C_VEL
LIN {X 0,Y 501.662,Z 658.288,A -85,B 0,C 180,E1 -13847.296,E2 -13847.296} C_VEL
LIN {X 0,Y 500.879,Z 667.451,A -85,B 0,C 180,E1 -13848.401,E2 -13848.401} C_VEL
LIN {X 0,Y 500.146,Z 676.482,A -85,B 0,C 180,E1 -13849.714,E2 -13849.714} C_VEL
LIN {X 0,Y 499.362,Z 684.427,A -85,B 0,C 180,E1 -13851.124,E2 -13851.124} C_VEL
LIN {X 0,Y 498.945,Z 689.973,A -85,B 0,C 180,E1 -13852.336,E2 -13852.336} C_VEL
LIN {X 0,Y 498.528,Z 695.78,A -85,B 0,C 180,E1 -13853.951,E2 -13853.951} C_VEL
LIN {X 0,Y 498.332,Z 699.057,A -85,B 0,C 180,E1 -13855.162,E2 -13855.162} C_VEL
LIN {X 0,Y 498.193,Z 702.078,A -85,B 0,C 180,E1 -13856.776,E2 -13856.776} C_VEL
LIN {X 0,Y 498.127,Z 703.645,A -85,B 0,C 180,E1 -13858.389,E2 -13858.389} C_VEL
LIN {X 0,Y 498.131,Z 703.778,A -85,B 0,C 180,E1 -13860,E2 -13860} C_VEL
LIN {X 0,Y 498.124,Z 702.446,A -85,B 0,C 180,E1 -13861.612,E2 -13861.612} C_VEL
LIN {X 0,Y 498.145,Z 699.621,A -85,B 0,C 180,E1 -13863.224,E2 -13863.224} C_VEL
LIN {X 0,Y 498.252,Z 695.262,A -85,B 0,C 180,E1 -13864.839,E2 -13864.839} C_VEL
LIN {X 0,Y 498.355,Z 690.898,A -85,B 0,C 180,E1 -13866.051,E2 -13866.051} C_VEL
LIN {X 0,Y 498.599,Z 684.48,A -85,B 0,C 180,E1 -13867.467,E2 -13867.467} C_VEL
LIN {X 0,Y 498.919,Z 676.454,A -85,B 0,C 180,E1 -13868.884,E2 -13868.884} C_VEL
LIN {X 0,Y 499.33,Z 668.044,A -85,B 0,C 180,E1 -13870.099,E2 -13870.099} C_VEL
LIN {X 0,Y 499.878,Z 657.914,A -85,B 0,C 180,E1 -13871.313,E2 -13871.313} C_VEL
LIN {X 0,Y 500.404,Z 646.574,A -85,B 0,C 180,E1 -13872.428,E2 -13872.428} C_VEL
LIN {X 0,Y 501.05,Z 633.995,A -85,B 0,C 180,E1 -13873.439,E2 -13873.439} C_VEL
LIN {X 0,Y 501.709,Z 621.654,A -85,B 0,C 180,E1 -13874.245,E2 -13874.245} C_VEL
LIN {X 0,Y 502.343,Z 608.152,A -85,B 0,C 180,E1 -13874.949,E2 -13874.949} C_VEL
LIN {X 0,Y 502.79,Z 593.358,A -85,B 0,C 180,E1 -13875.53,E2 -13875.53} C_VEL
LIN {X 0,Y 503.248,Z 578.752,A -85,B 0,C 180,E1 -13875.93,E2 -13875.93} C_VEL
LIN {X 0,Y 505.296,Z 464.322,A -85,B 0,C 180,E1 -13877.975,E2 -13877.975} C_VEL
LIN {X 0,Y 502.527,Z 439.528,A -85,B 0,C 180,E1 -13878.522,E2 -13878.522} C_VEL
LIN {X 0,Y 503.877,Z 408.458,A -85,B 0,C 180,E1 -13882.045,E2 -13882.045} C_VEL
LIN {X 0,Y 505.172,Z 382.297,A -85,B 0,C 180,E1 -13885.018,E2 -13885.018} C_VEL
LIN {X 0,Y 506.034,Z 363.377,A -85,B 0,C 180,E1 -13887.18,E2 -13887.18} C_VEL
LIN {X 0,Y 501.519,Z 342.771,A -85,B 0,C 180,E1 -13889.771,E2 -13889.771} C_VEL
LIN {X 0,Y 499.895,Z 335.773,A -85,B 0,C 180,E1 -13890.672,E2 -13890.672} C_VEL
LIN {X 0,Y 499.883,Z 335.777,A -85,B 0,C 180,E1 -13893.126,E2 -13893.126} C_VEL
LIN {X 0,Y 499.909,Z 335.768,A -85,B 0,C 180,E1 -13896.05,E2 -13896.05} C_VEL
LIN {X 0,Y 499.888,Z 335.773,A -85,B 0,C 180,E1 -13899.587,E2 -13899.587} C_VEL
LIN {X 0,Y 499.855,Z 335.774,A -85,B 0,C 180,E1 -13902.27,E2 -13902.27} C_VEL
LIN {X 0,Y 499.894,Z 335.771,A -85,B 0,C 180,E1 -13905.525,E2 -13905.525} C_VEL
LIN {X 0,Y 499.884,Z 335.779,A -85,B 0,C 180,E1 -13908.809,E2 -13908.809} C_VEL
LIN {X 0,Y 499.848,Z 335.775,A -85,B 0,C 180,E1 -13911.697,E2 -13911.697} C_VEL
LIN {X 0,Y 499.896,Z 335.773,A -85,B 0,C 180,E1 -13914.36,E2 -13914.36} C_VEL
LIN {X 0,Y 499.856,Z 335.775,A -85,B 0,C 180,E1 -13917.223,E2 -13917.223} C_VEL
LIN {X 0,Y 499.887,Z 335.776,A -85,B 0,C 180,E1 -13920.314,E2 -13920.314} C_VEL
LIN {X 0,Y 499.885,Z 335.778,A -85,B 0,C 180,E1 -13922.458,E2 -13922.458} C_VEL
LIN {X 0,Y 499.887,Z 335.771,A -85,B 0,C 180,E1 -13925.615,E2 -13925.615} C_VEL
LIN {X 0,Y 499.922,Z 335.769,A -85,B 0,C 180,E1 -13928.636,E2 -13928.636} C_VEL
LIN {X 0,Y 499.893,Z 335.77,A -85,B 0,C 180,E1 -13931.2,E2 -13931.2} C_VEL
LIN {X 0,Y 499.899,Z 335.773,A -85,B 0,C 180,E1 -13933.726,E2 -13933.726} C_VEL
LIN {X 0,Y 499.938,Z 335.767,A -85,B 0,C 180,E1 -13936.463,E2 -13936.463} C_VEL
LIN {X 0,Y 506.508,Z 354.385,A -85,B 0,C 180,E1 -13936.977,E2 -13936.977} C_VEL
LIN {X 0,Y 505.596,Z 453.119,A -85,B 0,C 180,E1 -13938.386,E2 -13938.386} C_VEL
LIN {X 0,Y 505.488,Z 467.431,A -85,B 0,C 180,E1 -13938.713,E2 -13938.713} C_VEL
LIN {X 0,Y 505.195,Z 481.83,A -85,B 0,C 180,E1 -13939.212,E2 -13939.212} C_VEL
LIN {X 0,Y 505.101,Z 484.521,A -85,B 0,C 180,E1 -13939.327,E2 -13939.327} C_VEL
LIN {X 0,Y 504.358,Z 490.1,A -85,B 0,C 180,E1 -13939.566,E2 -13939.566} C_VEL
LIN {X 0,Y 501.237,Z 498.903,A -85,B 0,C 180,E1 -13939.947,E2 -13939.947} C_VEL
LIN {X 0,Y 498.038,Z 507.428,A -85,B 0,C 180,E1 -13940.385,E2 -13940.385} C_VEL
LIN {X 0,Y 497.139,Z 512.4,A -85,B 0,C 180,E1 -13940.719,E2 -13940.719} C_VEL
LIN {X 0,Y 496.46,Z 524.153,A -85,B 0,C 180,E1 -13941.685,E2 -13941.685} C_VEL
LIN {X 0,Y 495.649,Z 534.274,A -85,B 0,C 180,E1 -13942.693,E2 -13942.693} C_VEL
LIN {X 0,Y 494.812,Z 544.352,A -85,B 0,C 180,E1 -13943.906,E2 -13943.906} C_VEL
LIN {X 0,Y 494.182,Z 552.674,A -85,B 0,C 180,E1 -13945.122,E2 -13945.122} C_VEL
LIN {X 0,Y 493.567,Z 560.632,A -85,B 0,C 180,E1 -13946.542,E2 -13946.542} C_VEL
LIN {X 0,Y 493.121,Z 567.049,A -85,B 0,C 180,E1 -13947.965,E2 -13947.965} C_VEL
LIN {X 0,Y 492.568,Z 572.773,A -85,B 0,C 180,E1 -13949.593,E2 -13949.593} C_VEL
LIN {X 0,Y 492.41,Z 576.069,A -85,B 0,C 180,E1 -13950.815,E2 -13950.815} C_VEL
LIN {X 0,Y 492.329,Z 579.167,A -85,B 0,C 180,E1 -13952.446,E2 -13952.446} C_VEL
LIN {X 0,Y 492.193,Z 580.955,A -85,B 0,C 180,E1 -13954.081,E2 -13954.081} C_VEL
LIN {X 0,Y 492.309,Z 581.434,A -85,B 0,C 180,E1 -13955.716,E2 -13955.716} C_VEL
LIN {X 0,Y 492.43,Z 580.634,A -85,B 0,C 180,E1 -13957.355,E2 -13957.355} C_VEL
LIN {X 0,Y 492.669,Z 578.519,A -85,B 0,C 180,E1 -13958.998,E2 -13958.998} C_VEL
LIN {X 0,Y 493.168,Z 575.014,A -85,B 0,C 180,E1 -13960.64,E2 -13960.64} C_VEL
LIN {X 0,Y 493.696,Z 570.029,A -85,B 0,C 180,E1 -13962.288,E2 -13962.288} C_VEL
LIN {X 0,Y 494.298,Z 565.164,A -85,B 0,C 180,E1 -13963.522,E2 -13963.522} C_VEL
LIN {X 0,Y 495.052,Z 558.17,A -85,B 0,C 180,E1 -13964.965,E2 -13964.965} C_VEL
LIN {X 0,Y 496.021,Z 549.475,A -85,B 0,C 180,E1 -13966.405,E2 -13966.405} C_VEL
LIN {X 0,Y 496.937,Z 540.333,A -85,B 0,C 180,E1 -13967.641,E2 -13967.641} C_VEL
LIN {X 0,Y 497.816,Z 530.179,A -85,B 0,C 180,E1 -13968.776,E2 -13968.776} C_VEL
LIN {X 0,Y 498.634,Z 519.634,A -85,B 0,C 180,E1 -13969.751,E2 -13969.751} C_VEL
LIN {X 0,Y 499.552,Z 508.011,A -85,B 0,C 180,E1 -13970.628,E2 -13970.628} C_VEL
LIN {X 0,Y 500.264,Z 496.261,A -85,B 0,C 180,E1 -13971.349,E2 -13971.349} C_VEL
LIN {X 0,Y 500.686,Z 483.408,A -85,B 0,C 180,E1 -13971.977,E2 -13971.977} C_VEL
LIN {X 0,Y 501.115,Z 469.05,A -85,B 0,C 180,E1 -13972.487,E2 -13972.487} C_VEL
LIN {X 0,Y 501.283,Z 456.786,A -85,B 0,C 180,E1 -13972.788,E2 -13972.788} C_VEL
LIN {X 0,Y 502.414,Z 359.793,A -85,B 0,C 180,E1 -13974.212,E2 -13974.212} C_VEL
LIN {X 0,Y 493.751,Z 339.443,A -85,B 0,C 180,E1 -13974.929,E2 -13974.929} C_VEL
LIN {X 0,Y 492.789,Z 336.666,A -85,B 0,C 180,E1 -13975.047,E2 -13975.047} C_VEL
LIN {X 0,Y 492.814,Z 336.655,A -85,B 0,C 180,E1 -13977.972,E2 -13977.972} C_VEL
LIN {X 0,Y 492.797,Z 336.658,A -85,B 0,C 180,E1 -13980.777,E2 -13980.777} C_VEL
LIN {X 0,Y 492.758,Z 336.662,A -85,B 0,C 180,E1 -13983.668,E2 -13983.668} C_VEL
LIN {X 0,Y 492.768,Z 336.662,A -85,B 0,C 180,E1 -13986.656,E2 -13986.656} C_VEL
LIN {X 0,Y 492.781,Z 336.661,A -85,B 0,C 180,E1 -13989.864,E2 -13989.864} C_VEL
LIN {X 0,Y 492.827,Z 336.653,A -85,B 0,C 180,E1 -13993.017,E2 -13993.017} C_VEL
LIN {X 0,Y 492.82,Z 336.655,A -85,B 0,C 180,E1 -13995.858,E2 -13995.858} C_VEL
LIN {X 0,Y 492.792,Z 336.654,A -85,B 0,C 180,E1 -13998.88,E2 -13998.88} C_VEL
LIN {X 0,Y 492.77,Z 336.655,A -85,B 0,C 180,E1 -14001.426,E2 -14001.426} C_VEL
LIN {X 0,Y 492.768,Z 336.641,A -85,B 0,C 180,E1 -14004.352,E2 -14004.352} C_VEL
LIN {X 0,Y 492.777,Z 336.655,A -85,B 0,C 180,E1 -14006.997,E2 -14006.997} C_VEL
LIN {X 0,Y 492.833,Z 336.651,A -85,B 0,C 180,E1 -14010.169,E2 -14010.169} C_VEL
LIN {X 0,Y 492.819,Z 336.649,A -85,B 0,C 180,E1 -14012.947,E2 -14012.947} C_VEL
LIN {X 0,Y 492.85,Z 336.65,A -85,B 0,C 180,E1 -14015.66,E2 -14015.66} C_VEL
LIN {X 0,Y 492.828,Z 336.647,A -85,B 0,C 180,E1 -14019.187,E2 -14019.187} C_VEL
LIN {X 0,Y 492.858,Z 336.653,A -85,B 0,C 180,E1 -14020.921,E2 -14020.921} C_VEL
LIN {X 0,Y 498.125,Z 354.538,A -85,B 0,C 180,E1 -14021.406,E2 -14021.406} C_VEL
LIN {X 0,Y 496.437,Z 455.866,A -85,B 0,C 180,E1 -14023.24,E2 -14023.24} C_VEL
LIN {X 0,Y 496.231,Z 470.819,A -85,B 0,C 180,E1 -14023.68,E2 -14023.68} C_VEL
LIN {X 0,Y 495.861,Z 484.931,A -85,B 0,C 180,E1 -14024.257,E2 -14024.257} C_VEL
LIN {X 0,Y 495.479,Z 497.85,A -85,B 0,C 180,E1 -14024.944,E2 -14024.944} C_VEL
LIN {X 0,Y 495.055,Z 510.243,A -85,B 0,C 180,E1 -14025.769,E2 -14025.769} C_VEL
LIN {X 0,Y 494.475,Z 522.826,A -85,B 0,C 180,E1 -14026.796,E2 -14026.796} C_VEL
LIN {X 0,Y 494.002,Z 533.611,A -85,B 0,C 180,E1 -14027.864,E2 -14027.864} C_VEL
LIN {X 0,Y 493.65,Z 542.838,A -85,B 0,C 180,E1 -14028.956,E2 -14028.956} C_VEL
LIN {X 0,Y 493.137,Z 551.58,A -85,B 0,C 180,E1 -14030.186,E2 -14030.186} C_VEL
LIN {X 0,Y 492.774,Z 559.911,A -85,B 0,C 180,E1 -14031.622,E2 -14031.622} C_VEL
LIN {X 0,Y 492.462,Z 566.604,A -85,B 0,C 180,E1 -14033.056,E2 -14033.056} C_VEL
LIN {X 0,Y 492.314,Z 571.225,A -85,B 0,C 180,E1 -14034.284,E2 -14034.284} C_VEL
LIN {X 0,Y 492.191,Z 575.893,A -85,B 0,C 180,E1 -14035.919,E2 -14035.919} C_VEL
LIN {X 0,Y 492.26,Z 579.035,A -85,B 0,C 180,E1 -14037.553,E2 -14037.553} C_VEL
LIN {X 0,Y 492.229,Z 580.751,A -85,B 0,C 180,E1 -14039.184,E2 -14039.184} C_VEL
LIN {X 0,Y 492.286,Z 581.01,A -85,B 0,C 180,E1 -14040.815,E2 -14040.815} C_VEL
LIN {X 0,Y 492.608,Z 579.833,A -85,B 0,C 180,E1 -14042.445,E2 -14042.445} C_VEL
LIN {X 0,Y 493.211,Z 577.206,A -85,B 0,C 180,E1 -14044.072,E2 -14044.072} C_VEL
LIN {X 0,Y 493.569,Z 574.258,A -85,B 0,C 180,E1 -14045.293,E2 -14045.293} C_VEL
LIN {X 0,Y 493.924,Z 570.437,A -85,B 0,C 180,E1 -14046.514,E2 -14046.514} C_VEL
LIN {X 0,Y 494.758,Z 565.056,A -85,B 0,C 180,E1 -14047.842,E2 -14047.842} C_VEL
LIN {X 0,Y 495.662,Z 557.372,A -85,B 0,C 180,E1 -14049.353,E2 -14049.353} C_VEL
LIN {X 0,Y 496.443,Z 549.737,A -85,B 0,C 180,E1 -14050.569,E2 -14050.569} C_VEL
LIN {X 0,Y 497.346,Z 540.512,A -85,B 0,C 180,E1 -14051.783,E2 -14051.783} C_VEL
LIN {X 0,Y 498.165,Z 530.338,A -85,B 0,C 180,E1 -14052.897,E2 -14052.897} C_VEL
LIN {X 0,Y 499.233,Z 518.372,A -85,B 0,C 180,E1 -14053.954,E2 -14053.954} C_VEL
LIN {X 0,Y 500.209,Z 505.579,A -85,B 0,C 180,E1 -14054.87,E2 -14054.87} C_VEL
LIN {X 0,Y 500.896,Z 492.665,A -85,B 0,C 180,E1 -14055.616,E2 -14055.616} C_VEL
LIN {X 0,Y 501.348,Z 478.443,A -85,B 0,C 180,E1 -14056.252,E2 -14056.252} C_VEL
LIN {X 0,Y 501.722,Z 463.415,A -85,B 0,C 180,E1 -14056.735,E2 -14056.735} C_VEL
LIN {X 0,Y 504.079,Z 388.869,A -85,B 0,C 180,E1 -14058.268,E2 -14058.268} C_VEL
LIN {X 0,Y 505.12,Z 361.689,A -85,B 0,C 180,E1 -14058.843,E2 -14058.843} C_VEL
LIN {X 0,Y 498.24,Z 347.359,A -85,B 0,C 180,E1 -14059.686,E2 -14059.686} C_VEL
LIN {X 0,Y 494.171,Z 339.938,A -85,B 0,C 180,E1 -14060.196,E2 -14060.196} C_VEL
LIN {X 0,Y 492.964,Z 337.197,A -85,B 0,C 180,E1 -14060.364,E2 -14060.364} C_VEL
LIN {X 0,Y 492.879,Z 336.65,A -85,B 0,C 180,E1 -14060.394,E2 -14060.394} C_VEL
LIN {X 0,Y 492.82,Z 336.66,A -85,B 0,C 180,E1 -14063.451,E2 -14063.451} C_VEL
LIN {X 0,Y 492.847,Z 336.654,A -85,B 0,C 180,E1 -14066.443,E2 -14066.443} C_VEL
LIN {X 0,Y 492.836,Z 336.652,A -85,B 0,C 180,E1 -14068.896,E2 -14068.896} C_VEL
LIN {X 0,Y 492.837,Z 336.652,A -85,B 0,C 180,E1 -14071.726,E2 -14071.726} C_VEL
LIN {X 0,Y 492.839,Z 336.648,A -85,B 0,C 180,E1 -14074.645,E2 -14074.645} C_VEL
LIN {X 0,Y 492.846,Z 336.645,A -85,B 0,C 180,E1 -14077.26,E2 -14077.26} C_VEL
LIN {X 0,Y 492.788,Z 336.652,A -85,B 0,C 180,E1 -14079.865,E2 -14079.865} C_VEL
LIN {X 0,Y 492.84,Z 336.649,A -85,B 0,C 180,E1 -14083.015,E2 -14083.015} C_VEL
LIN {X 0,Y 492.818,Z 336.65,A -85,B 0,C 180,E1 -14085.858,E2 -14085.858} C_VEL
LIN {X 0,Y 492.789,Z 336.662,A -85,B 0,C 180,E1 -14088.88,E2 -14088.88} C_VEL
LIN {X 0,Y 492.768,Z 336.66,A -85,B 0,C 180,E1 -14091.425,E2 -14091.425} C_VEL
LIN {X 0,Y 492.764,Z 336.665,A -85,B 0,C 180,E1 -14094.352,E2 -14094.352} C_VEL
LIN {X 0,Y 492.753,Z 336.664,A -85,B 0,C 180,E1 -14097.305,E2 -14097.305} C_VEL
LIN {X 0,Y 492.827,Z 336.714,A -85,B 0,C 180,E1 -14098.454,E2 -14098.454} C_VEL
LIN {X 0,Y 496.742,Z 353.104,A -85,B 0,C 180,E1 -14100.956,E2 -14100.956} C_VEL
LIN {X 0,Y 498.772,Z 362.888,A -85,B 0,C 180,E1 -14102.391,E2 -14102.391} C_VEL
LIN {X 0,Y 498.824,Z 366.256,A -85,B 0,C 180,E1 -14102.847,E2 -14102.847} C_VEL
LIN {X 0,Y 497.001,Z 389.583,A -85,B 0,C 180,E1 -14105.876,E2 -14105.876} C_VEL
LIN {X 0,Y 495.337,Z 414.926,A -85,B 0,C 180,E1 -14109.138,E2 -14109.138} C_VEL
LIN {X 0,Y 498.878,Z 439.75,A -85,B 0,C 180,E1 -14109.986,E2 -14109.986} C_VEL
LIN {X 0,Y 501.266,Z 468.085,A -85,B 0,C 180,E1 -14110.793,E2 -14110.793} C_VEL
LIN {X 0,Y 501.244,Z 474.066,A -85,B 0,C 180,E1 -14110.93,E2 -14110.93} C_VEL
LIN {X 0,Y 500.712,Z 490.613,A -85,B 0,C 180,E1 -14111.258,E2 -14111.258} C_VEL
LIN {X 0,Y 499.703,Z 561.666,A -85,B 0,C 180,E1 -14112.302,E2 -14112.302} C_VEL
LIN {X 0,Y 499.003,Z 576.374,A -85,B 0,C 180,E1 -14112.681,E2 -14112.681} C_VEL
LIN {X 0,Y 497.995,Z 590.16,A -85,B 0,C 180,E1 -14113.195,E2 -14113.195} C_VEL
LIN {X 0,Y 497.024,Z 602.991,A -85,B 0,C 180,E1 -14113.839,E2 -14113.839} C_VEL
LIN {X 0,Y 495.89,Z 615.605,A -85,B 0,C 180,E1 -14114.642,E2 -14114.642} C_VEL
LIN {X 0,Y 494.816,Z 627.142,A -85,B 0,C 180,E1 -14115.552,E2 -14115.552} C_VEL
LIN {X 0,Y 493.901,Z 636.789,A -85,B 0,C 180,E1 -14116.467,E2 -14116.467} C_VEL
LIN {X 0,Y 493.335,Z 644.632,A -85,B 0,C 180,E1 -14117.287,E2 -14117.287} C_VEL
LIN {X 0,Y 492.799,Z 655.82,A -85,B 0,C 180,E1 -14118.314,E2 -14118.314} C_VEL
LIN {X 0,Y 492.282,Z 666.859,A -85,B 0,C 180,E1 -14119.548,E2 -14119.548} C_VEL
LIN {X 0,Y 491.867,Z 675.949,A -85,B 0,C 180,E1 -14120.781,E2 -14120.781} C_VEL
LIN {X 0,Y 491.485,Z 684.615,A -85,B 0,C 180,E1 -14122.219,E2 -14122.219} C_VEL
LIN {X 0,Y 491.327,Z 690.619,A -85,B 0,C 180,E1 -14123.451,E2 -14123.451} C_VEL
LIN {X 0,Y 491.255,Z 695.5,A -85,B 0,C 180,E1 -14124.682,E2 -14124.682} C_VEL
LIN {X 0,Y 491.16,Z 699.38,A -85,B 0,C 180,E1 -14125.911,E2 -14125.911} C_VEL
LIN {X 0,Y 491.108,Z 703.117,A -85,B 0,C 180,E1 -14127.548,E2 -14127.548} C_VEL
LIN {X 0,Y 491.121,Z 705.336,A -85,B 0,C 180,E1 -14129.183,E2 -14129.183} C_VEL
LIN {X 0,Y 491.121,Z 706.072,A -85,B 0,C 180,E1 -14130.817,E2 -14130.817} C_VEL
LIN {X 0,Y 491.115,Z 705.306,A -85,B 0,C 180,E1 -14132.452,E2 -14132.452} C_VEL
LIN {X 0,Y 491.167,Z 703.075,A -85,B 0,C 180,E1 -14134.089,E2 -14134.089} C_VEL
LIN {X 0,Y 491.4,Z 699.347,A -85,B 0,C 180,E1 -14135.726,E2 -14135.726} C_VEL
LIN {X 0,Y 491.721,Z 694.016,A -85,B 0,C 180,E1 -14137.366,E2 -14137.366} C_VEL
LIN {X 0,Y 492.119,Z 688.817,A -85,B 0,C 180,E1 -14138.595,E2 -14138.595} C_VEL
LIN {X 0,Y 492.761,Z 681.381,A -85,B 0,C 180,E1 -14140.028,E2 -14140.028} C_VEL
LIN {X 0,Y 493.565,Z 672.121,A -85,B 0,C 180,E1 -14141.46,E2 -14141.46} C_VEL
LIN {X 0,Y 494.403,Z 662.422,A -85,B 0,C 180,E1 -14142.685,E2 -14142.685} C_VEL
LIN {X 0,Y 495.412,Z 651.72,A -85,B 0,C 180,E1 -14143.803,E2 -14143.803} C_VEL
LIN {X 0,Y 496.257,Z 641.241,A -85,B 0,C 180,E1 -14144.718,E2 -14144.718} C_VEL
LIN {X 0,Y 497.339,Z 628.559,A -85,B 0,C 180,E1 -14145.626,E2 -14145.626} C_VEL
LIN {X 0,Y 498.329,Z 614.485,A -85,B 0,C 180,E1 -14146.432,E2 -14146.432} C_VEL
LIN {X 0,Y 499.211,Z 600.709,A -85,B 0,C 180,E1 -14147.031,E2 -14147.031} C_VEL
LIN {X 0,Y 499.956,Z 586.747,A -85,B 0,C 180,E1 -14147.478,E2 -14147.478} C_VEL
LIN {X 0,Y 501.218,Z 553.125,A -85,B 0,C 180,E1 -14148.181,E2 -14148.181} C_VEL
LIN {X 0,Y 504.336,Z 470.986,A -85,B 0,C 180,E1 -14149.917,E2 -14149.917} C_VEL
LIN {X 0,Y 503.07,Z 452.076,A -85,B 0,C 180,E1 -14150.473,E2 -14150.473} C_VEL
LIN {X 0,Y 501.146,Z 435.706,A -85,B 0,C 180,E1 -14151.041,E2 -14151.041} C_VEL
LIN {X 0,Y 499.568,Z 415.561,A -85,B 0,C 180,E1 -14152.127,E2 -14152.127} C_VEL
LIN {X 0,Y 497.654,Z 394.655,A -85,B 0,C 180,E1 -14153.429,E2 -14153.429} C_VEL
LIN {X 0,Y 496.219,Z 378.916,A -85,B 0,C 180,E1 -14154.553,E2 -14154.553} C_VEL
LIN {X 0,Y 497.446,Z 360.077,A -85,B 0,C 180,E1 -14156.953,E2 -14156.953} C_VEL
LIN {X 0,Y 495.106,Z 347.119,A -85,B 0,C 180,E1 -14158.751,E2 -14158.751} C_VEL
LIN {X 0,Y 492.861,Z 336.649,A -85,B 0,C 180,E1 -14160.256,E2 -14160.256} C_VEL
LIN {X 0,Y 492.753,Z 336.662,A -85,B 0,C 180,E1 -14163.668,E2 -14163.668} C_VEL
LIN {X 0,Y 492.762,Z 336.662,A -85,B 0,C 180,E1 -14166.656,E2 -14166.656} C_VEL
LIN {X 0,Y 492.776,Z 336.657,A -85,B 0,C 180,E1 -14169.864,E2 -14169.864} C_VEL
LIN {X 0,Y 492.824,Z 336.656,A -85,B 0,C 180,E1 -14173.017,E2 -14173.017} C_VEL
LIN {X 0,Y 492.813,Z 336.658,A -85,B 0,C 180,E1 -14175.857,E2 -14175.857} C_VEL
LIN {X 0,Y 492.78,Z 336.658,A -85,B 0,C 180,E1 -14178.881,E2 -14178.881} C_VEL
LIN {X 0,Y 492.781,Z 336.66,A -85,B 0,C 180,E1 -14181.424,E2 -14181.424} C_VEL
LIN {X 0,Y 492.857,Z 336.781,A -85,B 0,C 180,E1 -14184.246,E2 -14184.246} C_VEL
LIN {X 0,Y 497.561,Z 348.442,A -85,B 0,C 180,E1 -14186.7,E2 -14186.7} C_VEL
LIN {X 0,Y 501.192,Z 358.927,A -85,B 0,C 180,E1 -14188.628,E2 -14188.628} C_VEL
LIN {X 0,Y 503.952,Z 368.913,A -85,B 0,C 180,E1 -14190.278,E2 -14190.278} C_VEL
LIN {X 0,Y 505.376,Z 376.53,A -85,B 0,C 180,E1 -14191.423,E2 -14191.423} C_VEL
LIN {X 0,Y 503.38,Z 399.899,A -85,B 0,C 180,E1 -14194.225,E2 -14194.225} C_VEL
LIN {X 0,Y 501.054,Z 429.098,A -85,B 0,C 180,E1 -14197.678,E2 -14197.678} C_VEL
LIN {X 0,Y 500.334,Z 439.982,A -85,B 0,C 180,E1 -14198.933,E2 -14198.933} C_VEL
LIN {X 0,Y 503.607,Z 457.823,A -85,B 0,C 180,E1 -14199.616,E2 -14199.616} C_VEL
LIN {X 0,Y 504.934,Z 468.494,A -85,B 0,C 180,E1 -14199.965,E2 -14199.965} C_VEL
LIN {X 0,Y 501.83,Z 549.737,A -85,B 0,C 180,E1 -14201.655,E2 -14201.655} C_VEL
LIN {X 0,Y 500.582,Z 583.035,A -85,B 0,C 180,E1 -14202.35,E2 -14202.35} C_VEL
LIN {X 0,Y 499.786,Z 596.883,A -85,B 0,C 180,E1 -14202.79,E2 -14202.79} C_VEL
LIN {X 0,Y 498.841,Z 610.483,A -85,B 0,C 180,E1 -14203.376,E2 -14203.376} C_VEL
LIN {X 0,Y 498.016,Z 623.134,A -85,B 0,C 180,E1 -14204.082,E2 -14204.082} C_VEL
LIN {X 0,Y 496.992,Z 634.945,A -85,B 0,C 180,E1 -14204.887,E2 -14204.887} C_VEL
LIN {X 0,Y 495.908,Z 647.129,A -85,B 0,C 180,E1 -14205.898,E2 -14205.898} C_VEL
LIN {X 0,Y 494.959,Z 657.23,A -85,B 0,C 180,E1 -14206.913,E2 -14206.913} C_VEL
LIN {X 0,Y 494.039,Z 666.607,A -85,B 0,C 180,E1 -14208.036,E2 -14208.036} C_VEL
LIN {X 0,Y 493.323,Z 675.775,A -85,B 0,C 180,E1 -14209.364,E2 -14209.364} C_VEL
LIN {X 0,Y 492.461,Z 683.841,A -85,B 0,C 180,E1 -14210.793,E2 -14210.793} C_VEL
LIN {X 0,Y 491.913,Z 690.324,A -85,B 0,C 180,E1 -14212.226,E2 -14212.226} C_VEL
LIN {X 0,Y 491.485,Z 696.065,A -85,B 0,C 180,E1 -14213.864,E2 -14213.864} C_VEL
LIN {X 0,Y 491.253,Z 699.266,A -85,B 0,C 180,E1 -14215.093,E2 -14215.093} C_VEL
LIN {X 0,Y 491.112,Z 702.216,A -85,B 0,C 180,E1 -14216.73,E2 -14216.73} C_VEL
LIN {X 0,Y 491.032,Z 703.716,A -85,B 0,C 180,E1 -14218.365,E2 -14218.365} C_VEL
LIN {X 0,Y 491.048,Z 703.766,A -85,B 0,C 180,E1 -14220,E2 -14220} C_VEL
LIN {X 0,Y 491.028,Z 702.332,A -85,B 0,C 180,E1 -14221.635,E2 -14221.635} C_VEL
LIN {X 0,Y 491.072,Z 699.428,A -85,B 0,C 180,E1 -14223.271,E2 -14223.271} C_VEL
LIN {X 0,Y 491.154,Z 694.983,A -85,B 0,C 180,E1 -14224.909,E2 -14224.909} C_VEL
LIN {X 0,Y 491.267,Z 690.527,A -85,B 0,C 180,E1 -14226.139,E2 -14226.139} C_VEL
LIN {X 0,Y 491.541,Z 684.003,A -85,B 0,C 180,E1 -14227.575,E2 -14227.575} C_VEL
LIN {X 0,Y 491.863,Z 675.855,A -85,B 0,C 180,E1 -14229.013,E2 -14229.013} C_VEL
LIN {X 0,Y 492.319,Z 667.313,A -85,B 0,C 180,E1 -14230.244,E2 -14230.244} C_VEL
LIN {X 0,Y 492.847,Z 656.962,A -85,B 0,C 180,E1 -14231.477,E2 -14231.477} C_VEL
LIN {X 0,Y 493.431,Z 645.415,A -85,B 0,C 180,E1 -14232.607,E2 -14232.607} C_VEL
LIN {X 0,Y 494.093,Z 632.595,A -85,B 0,C 180,E1 -14233.632,E2 -14233.632} C_VEL
LIN {X 0,Y 494.728,Z 619.931,A -85,B 0,C 180,E1 -14234.45,E2 -14234.45} C_VEL
LIN {X 0,Y 495.372,Z 605.804,A -85,B 0,C 180,E1 -14235.164,E2 -14235.164} C_VEL
LIN {X 0,Y 495.842,Z 590.994,A -85,B 0,C 180,E1 -14235.727,E2 -14235.727} C_VEL
LIN {X 0,Y 496.298,Z 576.524,A -85,B 0,C 180,E1 -14236.106,E2 -14236.106} C_VEL
LIN {X 0,Y 498.407,Z 465.785,A -85,B 0,C 180,E1 -14238.124,E2 -14238.124} C_VEL
LIN {X 0,Y 495.537,Z 439.495,A -85,B 0,C 180,E1 -14238.716,E2 -14238.716} C_VEL
LIN {X 0,Y 496.853,Z 411.308,A -85,B 0,C 180,E1 -14241.937,E2 -14241.937} C_VEL
LIN {X 0,Y 498.162,Z 385.051,A -85,B 0,C 180,E1 -14244.95,E2 -14244.95} C_VEL
LIN {X 0,Y 499.065,Z 366.024,A -85,B 0,C 180,E1 -14247.139,E2 -14247.139} C_VEL
LIN {X 0,Y 498.42,Z 361.423,A -85,B 0,C 180,E1 -14247.704,E2 -14247.704} C_VEL
LIN {X 0,Y 494.13,Z 342.203,A -85,B 0,C 180,E1 -14250.152,E2 -14250.152} C_VEL
LIN {X 0,Y 492.862,Z 336.651,A -85,B 0,C 180,E1 -14250.887,E2 -14250.887} C_VEL
LIN {X 0,Y 492.829,Z 336.653,A -85,B 0,C 180,E1 -14253.663,E2 -14253.663} C_VEL
LIN {X 0,Y 492.839,Z 336.649,A -85,B 0,C 180,E1 -14256.65,E2 -14256.65} C_VEL
LIN {X 0,Y 492.834,Z 336.649,A -85,B 0,C 180,E1 -14259.872,E2 -14259.872} C_VEL
LIN {X 0,Y 492.846,Z 336.656,A -85,B 0,C 180,E1 -14263.015,E2 -14263.015} C_VEL
LIN {X 0,Y 492.844,Z 336.647,A -85,B 0,C 180,E1 -14265.861,E2 -14265.861} C_VEL
LIN {X 0,Y 492.852,Z 336.65,A -85,B 0,C 180,E1 -14269.175,E2 -14269.175} C_VEL
LIN {X 0,Y 492.8,Z 336.656,A -85,B 0,C 180,E1 -14272.325,E2 -14272.325} C_VEL
LIN {X 0,Y 492.851,Z 336.651,A -85,B 0,C 180,E1 -14274.36,E2 -14274.36} C_VEL
LIN {X 0,Y 492.809,Z 336.653,A -85,B 0,C 180,E1 -14277.309,E2 -14277.309} C_VEL
LIN {X 0,Y 492.832,Z 336.653,A -85,B 0,C 180,E1 -14280.169,E2 -14280.169} C_VEL
LIN {X 0,Y 492.837,Z 336.65,A -85,B 0,C 180,E1 -14282.948,E2 -14282.948} C_VEL
LIN {X 0,Y 492.858,Z 336.647,A -85,B 0,C 180,E1 -14285.66,E2 -14285.66} C_VEL
LIN {X 0,Y 492.865,Z 336.652,A -85,B 0,C 180,E1 -14288.315,E2 -14288.315} C_VEL
LIN {X 0,Y 492.859,Z 336.646,A -85,B 0,C 180,E1 -14290.921,E2 -14290.921} C_VEL
LIN {X 0,Y 492.86,Z 336.647,A -85,B 0,C 180,E1 -14293.487,E2 -14293.487} C_VEL
LIN {X 0,Y 492.922,Z 336.753,A -85,B 0,C 180,E1 -14296.23,E2 -14296.23} C_VEL
LIN {X 0,Y 499.76,Z 355.931,A -85,B 0,C 180,E1 -14296.763,E2 -14296.763} C_VEL
LIN {X 0,Y 498.78,Z 452.101,A -85,B 0,C 180,E1 -14298.148,E2 -14298.148} C_VEL
LIN {X 0,Y 498.695,Z 466.207,A -85,B 0,C 180,E1 -14298.454,E2 -14298.454} C_VEL
LIN {X 0,Y 498.407,Z 479.91,A -85,B 0,C 180,E1 -14298.91,E2 -14298.91} C_VEL
LIN {X 0,Y 497.989,Z 492.242,A -85,B 0,C 180,E1 -14299.464,E2 -14299.464} C_VEL
LIN {X 0,Y 497.425,Z 504.503,A -85,B 0,C 180,E1 -14300.169,E2 -14300.169} C_VEL
LIN {X 0,Y 497.139,Z 512.4,A -85,B 0,C 180,E1 -14300.719,E2 -14300.719} C_VEL
LIN {X 0,Y 496.236,Z 517.368,A -85,B 0,C 180,E1 -14301.074,E2 -14301.074} C_VEL
LIN {X 0,Y 492.916,Z 525.257,A -85,B 0,C 180,E1 -14301.658,E2 -14301.658} C_VEL
LIN {X 0,Y 489.547,Z 532.725,A -85,B 0,C 180,E1 -14302.311,E2 -14302.311} C_VEL
LIN {X 0,Y 488.58,Z 537.032,A -85,B 0,C 180,E1 -14302.771,E2 -14302.771} C_VEL
LIN {X 0,Y 487.715,Z 546.898,A -85,B 0,C 180,E1 -14304.023,E2 -14304.023} C_VEL
LIN {X 0,Y 487.155,Z 554.909,A -85,B 0,C 180,E1 -14305.258,E2 -14305.258} C_VEL
LIN {X 0,Y 486.436,Z 562.607,A -85,B 0,C 180,E1 -14306.698,E2 -14306.698} C_VEL
LIN {X 0,Y 486.067,Z 567.993,A -85,B 0,C 180,E1 -14307.936,E2 -14307.936} C_VEL
LIN {X 0,Y 485.52,Z 573.675,A -85,B 0,C 180,E1 -14309.587,E2 -14309.587} C_VEL
LIN {X 0,Y 485.379,Z 576.932,A -85,B 0,C 180,E1 -14310.827,E2 -14310.827} C_VEL
LIN {X 0,Y 485.288,Z 579.994,A -85,B 0,C 180,E1 -14312.482,E2 -14312.482} C_VEL
LIN {X 0,Y 485.14,Z 581.749,A -85,B 0,C 180,E1 -14314.14,E2 -14314.14} C_VEL
LIN {X 0,Y 485.264,Z 582.194,A -85,B 0,C 180,E1 -14315.799,E2 -14315.799} C_VEL
LIN {X 0,Y 485.4,Z 581.359,A -85,B 0,C 180,E1 -14317.462,E2 -14317.462} C_VEL
LIN {X 0,Y 485.665,Z 579.209,A -85,B 0,C 180,E1 -14319.128,E2 -14319.128} C_VEL
LIN {X 0,Y 486.18,Z 575.668,A -85,B 0,C 180,E1 -14320.795,E2 -14320.795} C_VEL
LIN {X 0,Y 486.75,Z 570.643,A -85,B 0,C 180,E1 -14322.466,E2 -14322.466} C_VEL
LIN {X 0,Y 487.374,Z 565.736,A -85,B 0,C 180,E1 -14323.718,E2 -14323.718} C_VEL
LIN {X 0,Y 488.179,Z 558.694,A -85,B 0,C 180,E1 -14325.18,E2 -14325.18} C_VEL
LIN {X 0,Y 489.191,Z 549.946,A -85,B 0,C 180,E1 -14326.641,E2 -14326.641} C_VEL
LIN {X 0,Y 490.162,Z 540.729,A -85,B 0,C 180,E1 -14327.893,E2 -14327.893} C_VEL
LIN {X 0,Y 491.08,Z 530.48,A -85,B 0,C 180,E1 -14329.043,E2 -14329.043} C_VEL
LIN {X 0,Y 492,Z 519.129,A -85,B 0,C 180,E1 -14330.088,E2 -14330.088} C_VEL
LIN {X 0,Y 492.97,Z 506.501,A -85,B 0,C 180,E1 -14331.025,E2 -14331.025} C_VEL
LIN {X 0,Y 493.68,Z 494.163,A -85,B 0,C 180,E1 -14331.757,E2 -14331.757} C_VEL
LIN {X 0,Y 494.07,Z 483.023,A -85,B 0,C 180,E1 -14332.287,E2 -14332.287} C_VEL
LIN {X 0,Y 494.454,Z 468.936,A -85,B 0,C 180,E1 -14332.784,E2 -14332.784} C_VEL
LIN {X 0,Y 494.644,Z 455.329,A -85,B 0,C 180,E1 -14333.103,E2 -14333.103} C_VEL
LIN {X 0,Y 495.848,Z 361.627,A -85,B 0,C 180,E1 -14334.488,E2 -14334.488} C_VEL
LIN {X 0,Y 487.628,Z 342.397,A -85,B 0,C 180,E1 -14335.182,E2 -14335.182} C_VEL
LIN {X 0,Y 485.878,Z 338.272,A -85,B 0,C 180,E1 -14335.334,E2 -14335.334} C_VEL
LIN {X 0,Y 485.736,Z 337.543,A -85,B 0,C 180,E1 -14335.382,E2 -14335.382} C_VEL
LIN {X 0,Y 485.791,Z 337.53,A -85,B 0,C 180,E1 -14338.413,E2 -14338.413} C_VEL
LIN {X 0,Y 485.728,Z 337.535,A -85,B 0,C 180,E1 -14341.275,E2 -14341.275} C_VEL
LIN {X 0,Y 485.753,Z 337.536,A -85,B 0,C 180,E1 -14344.721,E2 -14344.721} C_VEL
LIN {X 0,Y 485.721,Z 337.538,A -85,B 0,C 180,E1 -14347.52,E2 -14347.52} C_VEL
LIN {X 0,Y 485.736,Z 337.541,A -85,B 0,C 180,E1 -14350.46,E2 -14350.46} C_VEL
LIN {X 0,Y 485.773,Z 337.536,A -85,B 0,C 180,E1 -14353.799,E2 -14353.799} C_VEL
LIN {X 0,Y 485.78,Z 337.536,A -85,B 0,C 180,E1 -14356.202,E2 -14356.202} C_VEL
LIN {X 0,Y 485.763,Z 337.532,A -85,B 0,C 180,E1 -14358.575,E2 -14358.575} C_VEL
LIN {X 0,Y 485.719,Z 337.526,A -85,B 0,C 180,E1 -14361.677,E2 -14361.677} C_VEL
LIN {X 0,Y 485.73,Z 337.522,A -85,B 0,C 180,E1 -14364.773,E2 -14364.773} C_VEL
LIN {X 0,Y 485.726,Z 337.54,A -85,B 0,C 180,E1 -14367.753,E2 -14367.753} C_VEL
LIN {X 0,Y 485.786,Z 337.525,A -85,B 0,C 180,E1 -14370.643,E2 -14370.643} C_VEL
LIN {X 0,Y 485.77,Z 337.529,A -85,B 0,C 180,E1 -14373.448,E2 -14373.448} C_VEL
LIN {X 0,Y 485.763,Z 337.533,A -85,B 0,C 180,E1 -14376.187,E2 -14376.187} C_VEL
LIN {X 0,Y 485.813,Z 337.529,A -85,B 0,C 180,E1 -14379.755,E2 -14379.755} C_VEL
LIN {X 0,Y 485.816,Z 337.53,A -85,B 0,C 180,E1 -14380.761,E2 -14380.761} C_VEL
LIN {X 0,Y 491.082,Z 355.05,A -85,B 0,C 180,E1 -14381.239,E2 -14381.239} C_VEL
LIN {X 0,Y 489.408,Z 456.87,A -85,B 0,C 180,E1 -14383.126,E2 -14383.126} C_VEL
LIN {X 0,Y 489.205,Z 472.489,A -85,B 0,C 180,E1 -14383.6,E2 -14383.6} C_VEL
LIN {X 0,Y 488.855,Z 486.705,A -85,B 0,C 180,E1 -14384.202,E2 -14384.202} C_VEL
LIN {X 0,Y 488.401,Z 499.92,A -85,B 0,C 180,E1 -14384.933,E2 -14384.933} C_VEL
LIN {X 0,Y 487.884,Z 513.454,A -85,B 0,C 180,E1 -14385.873,E2 -14385.873} C_VEL
LIN {X 0,Y 487.297,Z 525.657,A -85,B 0,C 180,E1 -14386.915,E2 -14386.915} C_VEL
LIN {X 0,Y 486.885,Z 536.382,A -85,B 0,C 180,E1 -14388.034,E2 -14388.034} C_VEL
LIN {X 0,Y 486.454,Z 545.805,A -85,B 0,C 180,E1 -14389.211,E2 -14389.211} C_VEL
LIN {X 0,Y 485.956,Z 555.426,A -85,B 0,C 180,E1 -14390.668,E2 -14390.668} C_VEL
LIN {X 0,Y 485.602,Z 563.216,A -85,B 0,C 180,E1 -14392.124,E2 -14392.124} C_VEL
LIN {X 0,Y 485.343,Z 568.609,A -85,B 0,C 180,E1 -14393.37,E2 -14393.37} C_VEL
LIN {X 0,Y 485.214,Z 572.982,A -85,B 0,C 180,E1 -14394.616,E2 -14394.616} C_VEL
LIN {X 0,Y 485.139,Z 576.435,A -85,B 0,C 180,E1 -14395.86,E2 -14395.86} C_VEL
LIN {X 0,Y 485.203,Z 579.692,A -85,B 0,C 180,E1 -14397.518,E2 -14397.518} C_VEL
LIN {X 0,Y 485.173,Z 581.526,A -85,B 0,C 180,E1 -14399.173,E2 -14399.173} C_VEL
LIN {X 0,Y 485.264,Z 581.912,A -85,B 0,C 180,E1 -14400.827,E2 -14400.827} C_VEL
LIN {X 0,Y 485.596,Z 580.835,A -85,B 0,C 180,E1 -14402.48,E2 -14402.48} C_VEL
LIN {X 0,Y 486.218,Z 578.302,A -85,B 0,C 180,E1 -14404.13,E2 -14404.13} C_VEL
LIN {X 0,Y 486.76,Z 574.315,A -85,B 0,C 180,E1 -14405.781,E2 -14405.781} C_VEL
LIN {X 0,Y 487.349,Z 569.784,A -85,B 0,C 180,E1 -14407.138,E2 -14407.138} C_VEL
LIN {X 0,Y 488.337,Z 563.169,A -85,B 0,C 180,E1 -14408.662,E2 -14408.662} C_VEL
LIN {X 0,Y 489.178,Z 555.309,A -85,B 0,C 180,E1 -14410.102,E2 -14410.102} C_VEL
LIN {X 0,Y 490.156,Z 547.051,A -85,B 0,C 180,E1 -14411.332,E2 -14411.332} C_VEL
LIN {X 0,Y 491.054,Z 537.105,A -85,B 0,C 180,E1 -14412.564,E2 -14412.564} C_VEL
LIN {X 0,Y 492.029,Z 527.055,A -85,B 0,C 180,E1 -14413.585,E2 -14413.585} C_VEL
LIN {X 0,Y 492.952,Z 516.626,A -85,B 0,C 180,E1 -14414.47,E2 -14414.47} C_VEL
LIN {X 0,Y 493.943,Z 503.773,A -85,B 0,C 180,E1 -14415.357,E2 -14415.357} C_VEL
LIN {X 0,Y 494.572,Z 489.7,A -85,B 0,C 180,E1 -14416.137,E2 -14416.137} C_VEL
LIN {X 0,Y 495.128,Z 475.682,A -85,B 0,C 180,E1 -14416.726,E2 -14416.726} C_VEL
LIN {X 0,Y 495.416,Z 460.877,A -85,B 0,C 180,E1 -14417.166,E2 -14417.166} C_VEL
LIN {X 0,Y 497.954,Z 388.611,A -85,B 0,C 180,E1 -14418.68,E2 -14418.68} C_VEL
LIN {X 0,Y 499.008,Z 364.005,A -85,B 0,C 180,E1 -14419.211,E2 -14419.211} C_VEL
LIN {X 0,Y 492.715,Z 350.93,A -85,B 0,C 180,E1 -14420.019,E2 -14420.019} C_VEL
LIN {X 0,Y 487.299,Z 341.027,A -85,B 0,C 180,E1 -14420.721,E2 -14420.721} C_VEL
LIN {X 0,Y 486.024,Z 338.509,A -85,B 0,C 180,E1 -14420.903,E2 -14420.903} C_VEL
LIN {X 0,Y 485.815,Z 337.531,A -85,B 0,C 180,E1 -14420.966,E2 -14420.966} C_VEL
LIN {X 0,Y 485.783,Z 337.535,A -85,B 0,C 180,E1 -14423.811,E2 -14423.811} C_VEL
LIN {X 0,Y 485.81,Z 337.531,A -85,B 0,C 180,E1 -14426.629,E2 -14426.629} C_VEL
LIN {X 0,Y 485.789,Z 337.531,A -85,B 0,C 180,E1 -14429.356,E2 -14429.356} C_VEL
LIN {X 0,Y 485.767,Z 337.532,A -85,B 0,C 180,E1 -14432.243,E2 -14432.243} C_VEL
LIN {X 0,Y 485.783,Z 337.526,A -85,B 0,C 180,E1 -14435.223,E2 -14435.223} C_VEL
LIN {X 0,Y 485.76,Z 337.526,A -85,B 0,C 180,E1 -14438.319,E2 -14438.319} C_VEL
LIN {X 0,Y 485.762,Z 337.53,A -85,B 0,C 180,E1 -14441.552,E2 -14441.552} C_VEL
LIN {X 0,Y 485.774,Z 337.526,A -85,B 0,C 180,E1 -14443.866,E2 -14443.866} C_VEL
LIN {X 0,Y 485.789,Z 337.53,A -85,B 0,C 180,E1 -14447.337,E2 -14447.337} C_VEL
LIN {X 0,Y 485.748,Z 337.538,A -85,B 0,C 180,E1 -14450.618,E2 -14450.618} C_VEL
LIN {X 0,Y 485.722,Z 337.539,A -85,B 0,C 180,E1 -14453.858,E2 -14453.858} C_VEL
LIN {X 0,Y 485.72,Z 337.543,A -85,B 0,C 180,E1 -14456.771,E2 -14456.771} C_VEL
LIN {X 0,Y 485.812,Z 337.734,A -85,B 0,C 180,E1 -14458.175,E2 -14458.175} C_VEL
LIN {X 0,Y 489.787,Z 354.176,A -85,B 0,C 180,E1 -14460.734,E2 -14460.734} C_VEL
LIN {X 0,Y 492.07,Z 365.811,A -85,B 0,C 180,E1 -14462.459,E2 -14462.459} C_VEL
LIN {X 0,Y 490.752,Z 382.367,A -85,B 0,C 180,E1 -14464.647,E2 -14464.647} C_VEL
LIN {X 0,Y 488.814,Z 408.942,A -85,B 0,C 180,E1 -14468.126,E2 -14468.126} C_VEL
LIN {X 0,Y 488.637,Z 412.842,A -85,B 0,C 180,E1 -14468.609,E2 -14468.609} C_VEL
LIN {X 0,Y 492.664,Z 440.679,A -85,B 0,C 180,E1 -14469.602,E2 -14469.602} C_VEL
LIN {X 0,Y 494.963,Z 468.706,A -85,B 0,C 180,E1 -14470.425,E2 -14470.425} C_VEL
LIN {X 0,Y 494.772,Z 479.129,A -85,B 0,C 180,E1 -14470.661,E2 -14470.661} C_VEL
LIN {X 0,Y 493.872,Z 504.161,A -85,B 0,C 180,E1 -14471.176,E2 -14471.176} C_VEL
LIN {X 0,Y 493.002,Z 560.743,A -85,B 0,C 180,E1 -14472.021,E2 -14472.021} C_VEL
LIN {X 0,Y 492.286,Z 575.481,A -85,B 0,C 180,E1 -14472.404,E2 -14472.404} C_VEL
LIN {X 0,Y 491.256,Z 589.332,A -85,B 0,C 180,E1 -14472.927,E2 -14472.927} C_VEL
LIN {X 0,Y 490.187,Z 602.684,A -85,B 0,C 180,E1 -14473.607,E2 -14473.607} C_VEL
LIN {X 0,Y 489.025,Z 615.205,A -85,B 0,C 180,E1 -14474.421,E2 -14474.421} C_VEL
LIN {X 0,Y 487.789,Z 627.849,A -85,B 0,C 180,E1 -14475.446,E2 -14475.446} C_VEL
LIN {X 0,Y 486.783,Z 638.231,A -85,B 0,C 180,E1 -14476.477,E2 -14476.477} C_VEL
LIN {X 0,Y 486.274,Z 645.776,A -85,B 0,C 180,E1 -14477.31,E2 -14477.31} C_VEL
LIN {X 0,Y 485.684,Z 656.769,A -85,B 0,C 180,E1 -14478.351,E2 -14478.351} C_VEL
LIN {X 0,Y 485.166,Z 667.656,A -85,B 0,C 180,E1 -14479.603,E2 -14479.603} C_VEL
LIN {X 0,Y 484.753,Z 676.618,A -85,B 0,C 180,E1 -14480.854,E2 -14480.854} C_VEL
LIN {X 0,Y 484.386,Z 685.123,A -85,B 0,C 180,E1 -14482.313,E2 -14482.313} C_VEL
LIN {X 0,Y 484.208,Z 691.907,A -85,B 0,C 180,E1 -14483.771,E2 -14483.771} C_VEL
LIN {X 0,Y 484.103,Z 696.568,A -85,B 0,C 180,E1 -14485.02,E2 -14485.02} C_VEL
LIN {X 0,Y 484.035,Z 701.2,A -85,B 0,C 180,E1 -14486.682,E2 -14486.682} C_VEL
LIN {X 0,Y 484.022,Z 704.258,A -85,B 0,C 180,E1 -14488.341,E2 -14488.341} C_VEL
LIN {X 0,Y 484.031,Z 705.817,A -85,B 0,C 180,E1 -14490,E2 -14490} C_VEL
LIN {X 0,Y 484.023,Z 705.902,A -85,B 0,C 180,E1 -14491.658,E2 -14491.658} C_VEL
LIN {X 0,Y 484.078,Z 704.49,A -85,B 0,C 180,E1 -14493.318,E2 -14493.318} C_VEL
LIN {X 0,Y 484.187,Z 701.591,A -85,B 0,C 180,E1 -14494.979,E2 -14494.979} C_VEL
LIN {X 0,Y 484.494,Z 697.154,A -85,B 0,C 180,E1 -14496.641,E2 -14496.641} C_VEL
LIN {X 0,Y 484.793,Z 692.738,A -85,B 0,C 180,E1 -14497.889,E2 -14497.889} C_VEL
LIN {X 0,Y 485.347,Z 686.261,A -85,B 0,C 180,E1 -14499.344,E2 -14499.344} C_VEL
LIN {X 0,Y 486.129,Z 678.192,A -85,B 0,C 180,E1 -14500.796,E2 -14500.796} C_VEL
LIN {X 0,Y 486.975,Z 668.838,A -85,B 0,C 180,E1 -14502.168,E2 -14502.168} C_VEL
LIN {X 0,Y 487.875,Z 659.623,A -85,B 0,C 180,E1 -14503.28,E2 -14503.28} C_VEL
LIN {X 0,Y 488.925,Z 648.354,A -85,B 0,C 180,E1 -14504.413,E2 -14504.413} C_VEL
LIN {X 0,Y 490.093,Z 635.842,A -85,B 0,C 180,E1 -14505.438,E2 -14505.438} C_VEL
LIN {X 0,Y 491.146,Z 623.568,A -85,B 0,C 180,E1 -14506.253,E2 -14506.253} C_VEL
LIN {X 0,Y 492.17,Z 609.213,A -85,B 0,C 180,E1 -14507.016,E2 -14507.016} C_VEL
LIN {X 0,Y 493.132,Z 594.117,A -85,B 0,C 180,E1 -14507.606,E2 -14507.606} C_VEL
LIN {X 0,Y 493.865,Z 579.382,A -85,B 0,C 180,E1 -14508.006,E2 -14508.006} C_VEL
LIN {X 0,Y 497.567,Z 487.477,A -85,B 0,C 180,E1 -14509.96,E2 -14509.96} C_VEL
LIN {X 0,Y 498.132,Z 470.797,A -85,B 0,C 180,E1 -14510.343,E2 -14510.343} C_VEL
LIN {X 0,Y 496.981,Z 452.906,A -85,B 0,C 180,E1 -14510.888,E2 -14510.888} C_VEL
LIN {X 0,Y 495.069,Z 436.661,A -85,B 0,C 180,E1 -14511.464,E2 -14511.464} C_VEL
LIN {X 0,Y 493.701,Z 417.615,A -85,B 0,C 180,E1 -14512.524,E2 -14512.524} C_VEL
LIN {X 0,Y 491.927,Z 395.956,A -85,B 0,C 180,E1 -14513.922,E2 -14513.922} C_VEL
LIN {X 0,Y 490.453,Z 379.5,A -85,B 0,C 180,E1 -14515.143,E2 -14515.143} C_VEL
LIN {X 0,Y 489.912,Z 370.512,A -85,B 0,C 180,E1 -14515.87,E2 -14515.87} C_VEL
LIN {X 0,Y 490.45,Z 360.322,A -85,B 0,C 180,E1 -14517.195,E2 -14517.195} C_VEL
LIN {X 0,Y 487.267,Z 344.173,A -85,B 0,C 180,E1 -14519.495,E2 -14519.495} C_VEL
LIN {X 0,Y 485.797,Z 337.528,A -85,B 0,C 180,E1 -14520.487,E2 -14520.487} C_VEL
LIN {X 0,Y 485.708,Z 337.544,A -85,B 0,C 180,E1 -14523.236,E2 -14523.236} C_VEL
LIN {X 0,Y 485.719,Z 337.536,A -85,B 0,C 180,E1 -14526.246,E2 -14526.246} C_VEL
LIN {X 0,Y 485.745,Z 337.531,A -85,B 0,C 180,E1 -14529.381,E2 -14529.381} C_VEL
LIN {X 0,Y 485.77,Z 337.535,A -85,B 0,C 180,E1 -14532.665,E2 -14532.665} C_VEL
LIN {X 0,Y 485.766,Z 337.536,A -85,B 0,C 180,E1 -14536.135,E2 -14536.135} C_VEL
LIN {X 0,Y 485.752,Z 337.533,A -85,B 0,C 180,E1 -14538.576,E2 -14538.576} C_VEL
LIN {X 0,Y 485.735,Z 337.536,A -85,B 0,C 180,E1 -14541.679,E2 -14541.679} C_VEL
LIN {X 0,Y 485.806,Z 337.6,A -85,B 0,C 180,E1 -14543.184,E2 -14543.184} C_VEL
LIN {X 0,Y 486.813,Z 340.433,A -85,B 0,C 180,E1 -14543.849,E2 -14543.849} C_VEL
LIN {X 0,Y 489.637,Z 346.862,A -85,B 0,C 180,E1 -14545.341,E2 -14545.341} C_VEL
LIN {X 0,Y 492.754,Z 354.878,A -85,B 0,C 180,E1 -14547.001,E2 -14547.001} C_VEL
LIN {X 0,Y 495.813,Z 364.237,A -85,B 0,C 180,E1 -14548.732,E2 -14548.732} C_VEL
LIN {X 0,Y 498.275,Z 373.809,A -85,B 0,C 180,E1 -14550.327,E2 -14550.327} C_VEL
LIN {X 0,Y 499.228,Z 379.566,A -85,B 0,C 180,E1 -14551.204,E2 -14551.204} C_VEL
LIN {X 0,Y 496.837,Z 405.052,A -85,B 0,C 180,E1 -14554.294,E2 -14554.294} C_VEL
LIN {X 0,Y 494.435,Z 433.716,A -85,B 0,C 180,E1 -14557.731,E2 -14557.731} C_VEL
LIN {X 0,Y 494.019,Z 439.975,A -85,B 0,C 180,E1 -14558.458,E2 -14558.458} C_VEL
LIN {X 0,Y 497.414,Z 458.451,A -85,B 0,C 180,E1 -14559.197,E2 -14559.197} C_VEL
LIN {X 0,Y 498.788,Z 469.704,A -85,B 0,C 180,E1 -14559.577,E2 -14559.577} C_VEL
LIN {X 0,Y 495.321,Z 554.377,A -85,B 0,C 180,E1 -14561.385,E2 -14561.385} C_VEL
LIN {X 0,Y 494.161,Z 583.185,A -85,B 0,C 180,E1 -14562.003,E2 -14562.003} C_VEL
LIN {X 0,Y 493.325,Z 596.773,A -85,B 0,C 180,E1 -14562.443,E2 -14562.443} C_VEL
LIN {X 0,Y 492.335,Z 610.456,A -85,B 0,C 180,E1 -14563.043,E2 -14563.043} C_VEL
LIN {X 0,Y 491.307,Z 624.707,A -85,B 0,C 180,E1 -14563.859,E2 -14563.859} C_VEL
LIN {X 0,Y 490.163,Z 637.553,A -85,B 0,C 180,E1 -14564.777,E2 -14564.777} C_VEL
LIN {X 0,Y 488.991,Z 649.197,A -85,B 0,C 180,E1 -14565.8,E2 -14565.8} C_VEL
LIN {X 0,Y 487.92,Z 659.842,A -85,B 0,C 180,E1 -14566.932,E2 -14566.932} C_VEL
LIN {X 0,Y 486.974,Z 669.543,A -85,B 0,C 180,E1 -14568.176,E2 -14568.176} C_VEL
LIN {X 0,Y 486.25,Z 677.575,A -85,B 0,C 180,E1 -14569.417,E2 -14569.417} C_VEL
LIN {X 0,Y 485.35,Z 685.331,A -85,B 0,C 180,E1 -14570.866,E2 -14570.866} C_VEL
LIN {X 0,Y 484.892,Z 690.71,A -85,B 0,C 180,E1 -14572.113,E2 -14572.113} C_VEL
LIN {X 0,Y 484.422,Z 696.364,A -85,B 0,C 180,E1 -14573.774,E2 -14573.774} C_VEL
LIN {X 0,Y 484.18,Z 699.487,A -85,B 0,C 180,E1 -14575.021,E2 -14575.021} C_VEL
LIN {X 0,Y 484.036,Z 702.367,A -85,B 0,C 180,E1 -14576.682,E2 -14576.682} C_VEL
LIN {X 0,Y 483.94,Z 703.787,A -85,B 0,C 180,E1 -14578.341,E2 -14578.341} C_VEL
LIN {X 0,Y 483.949,Z 703.73,A -85,B 0,C 180,E1 -14580,E2 -14580} C_VEL
LIN {X 0,Y 483.936,Z 702.212,A -85,B 0,C 180,E1 -14581.659,E2 -14581.659} C_VEL
LIN {X 0,Y 483.979,Z 699.22,A -85,B 0,C 180,E1 -14583.319,E2 -14583.319} C_VEL
LIN {X 0,Y 484.067,Z 694.678,A -85,B 0,C 180,E1 -14584.981,E2 -14584.981} C_VEL
LIN {X 0,Y 484.195,Z 690.122,A -85,B 0,C 180,E1 -14586.229,E2 -14586.229} C_VEL
LIN {X 0,Y 484.461,Z 683.487,A -85,B 0,C 180,E1 -14587.686,E2 -14587.686} C_VEL
LIN {X 0,Y 484.82,Z 675.205,A -85,B 0,C 180,E1 -14589.145,E2 -14589.145} C_VEL
LIN {X 0,Y 485.311,Z 666.502,A -85,B 0,C 180,E1 -14590.394,E2 -14590.394} C_VEL
LIN {X 0,Y 485.837,Z 655.95,A -85,B 0,C 180,E1 -14591.645,E2 -14591.645} C_VEL
LIN {X 0,Y 486.43,Z 644.203,A -85,B 0,C 180,E1 -14592.791,E2 -14592.791} C_VEL
LIN {X 0,Y 487.058,Z 632.538,A -85,B 0,C 180,E1 -14593.727,E2 -14593.727} C_VEL
LIN {X 0,Y 487.706,Z 619.865,A -85,B 0,C 180,E1 -14594.557,E2 -14594.557} C_VEL
LIN {X 0,Y 488.347,Z 605.739,A -85,B 0,C 180,E1 -14595.281,E2 -14595.281} C_VEL
LIN {X 0,Y 488.839,Z 591.161,A -85,B 0,C 180,E1 -14595.845,E2 -14595.845} C_VEL
LIN {X 0,Y 489.307,Z 575.969,A -85,B 0,C 180,E1 -14596.25,E2 -14596.25} C_VEL
LIN {X 0,Y 491.447,Z 465.962,A -85,B 0,C 180,E1 -14598.296,E2 -14598.296} C_VEL
LIN {X 0,Y 488.613,Z 439.459,A -85,B 0,C 180,E1 -14598.907,E2 -14598.907} C_VEL
LIN {X 0,Y 489.938,Z 410.395,A -85,B 0,C 180,E1 -14602.263,E2 -14602.263} C_VEL
LIN {X 0,Y 491.337,Z 383.963,A -85,B 0,C 180,E1 -14605.321,E2 -14605.321} C_VEL
LIN {X 0,Y 492.144,Z 366.894,A -85,B 0,C 180,E1 -14607.305,E2 -14607.305} C_VEL
LIN {X 0,Y 490.157,Z 356.654,A -85,B 0,C 180,E1 -14608.602,E2 -14608.602} C_VEL
LIN {X 0,Y 485.824,Z 337.528,A -85,B 0,C 180,E1 -14611.087,E2 -14611.087} C_VEL
LIN {X 0,Y 485.805,Z 337.524,A -85,B 0,C 180,E1 -14614.216,E2 -14614.216} C_VEL
LIN {X 0,Y 485.799,Z 337.532,A -85,B 0,C 180,E1 -14617.27,E2 -14617.27} C_VEL
LIN {X 0,Y 485.784,Z 337.528,A -85,B 0,C 180,E1 -14620.455,E2 -14620.455} C_VEL
LIN {X 0,Y 485.792,Z 337.526,A -85,B 0,C 180,E1 -14623.869,E2 -14623.869} C_VEL
LIN {X 0,Y 485.794,Z 337.526,A -85,B 0,C 180,E1 -14626.204,E2 -14626.204} C_VEL
LIN {X 0,Y 485.795,Z 337.526,A -85,B 0,C 180,E1 -14629.546,E2 -14629.546} C_VEL
LIN {X 0,Y 485.8,Z 337.533,A -85,B 0,C 180,E1 -14632.73,E2 -14632.73} C_VEL
LIN {X 0,Y 485.811,Z 337.524,A -85,B 0,C 180,E1 -14635.785,E2 -14635.785} C_VEL
LIN {X 0,Y 485.786,Z 337.532,A -85,B 0,C 180,E1 -14638.73,E2 -14638.73} C_VEL
LIN {X 0,Y 485.808,Z 337.524,A -85,B 0,C 180,E1 -14641.589,E2 -14641.589} C_VEL
LIN {X 0,Y 485.761,Z 337.538,A -85,B 0,C 180,E1 -14644.368,E2 -14644.368} C_VEL
LIN {X 0,Y 485.789,Z 337.526,A -85,B 0,C 180,E1 -14647.339,E2 -14647.339} C_VEL
LIN {X 0,Y 485.848,Z 337.522,A -85,B 0,C 180,E1 -14649.757,E2 -14649.757} C_VEL
LIN {X 0,Y 485.861,Z 337.522,A -85,B 0,C 180,E1 -14652.377,E2 -14652.377} C_VEL
LIN {X 0,Y 485.87,Z 337.524,A -85,B 0,C 180,E1 -14655.947,E2 -14655.947} C_VEL
LIN {X 0,Y 486.021,Z 338.39,A -85,B 0,C 180,E1 -14655.996,E2 -14655.996} C_VEL
LIN {X 0,Y 492.907,Z 357.155,A -85,B 0,C 180,E1 -14656.535,E2 -14656.535} C_VEL
LIN {X 0,Y 491.963,Z 454.023,A -85,B 0,C 180,E1 -14657.956,E2 -14657.956} C_VEL
LIN {X 0,Y 491.835,Z 468.579,A -85,B 0,C 180,E1 -14658.291,E2 -14658.291} C_VEL
LIN {X 0,Y 491.56,Z 481.808,A -85,B 0,C 180,E1 -14658.753,E2 -14658.753} C_VEL
LIN {X 0,Y 491.096,Z 493.878,A -85,B 0,C 180,E1 -14659.315,E2 -14659.315} C_VEL
LIN {X 0,Y 490.521,Z 505.96,A -85,B 0,C 180,E1 -14660.03,E2 -14660.03} C_VEL
LIN {X 0,Y 489.945,Z 518.381,A -85,B 0,C 180,E1 -14660.952,E2 -14660.952} C_VEL
LIN {X 0,Y 489.164,Z 529.633,A -85,B 0,C 180,E1 -14661.975,E2 -14661.975} C_VEL
LIN {X 0,Y 488.58,Z 537.032,A -85,B 0,C 180,E1 -14662.771,E2 -14662.771} C_VEL
LIN {X 0,Y 487.646,Z 541.221,A -85,B 0,C 180,E1 -14663.251,E2 -14663.251} C_VEL
LIN {X 0,Y 484.373,Z 547.769,A -85,B 0,C 180,E1 -14664.033,E2 -14664.033} C_VEL
LIN {X 0,Y 481.041,Z 553.927,A -85,B 0,C 180,E1 -14664.869,E2 -14664.869} C_VEL
LIN {X 0,Y 480.029,Z 557.328,A -85,B 0,C 180,E1 -14665.429,E2 -14665.429} C_VEL
LIN {X 0,Y 479.408,Z 563.592,A -85,B 0,C 180,E1 -14666.65,E2 -14666.65} C_VEL
LIN {X 0,Y 479.015,Z 568.936,A -85,B 0,C 180,E1 -14667.905,E2 -14667.905} C_VEL
LIN {X 0,Y 478.474,Z 574.576,A -85,B 0,C 180,E1 -14669.581,E2 -14669.581} C_VEL
LIN {X 0,Y 478.33,Z 577.795,A -85,B 0,C 180,E1 -14670.839,E2 -14670.839} C_VEL
LIN {X 0,Y 478.247,Z 580.82,A -85,B 0,C 180,E1 -14672.518,E2 -14672.518} C_VEL
LIN {X 0,Y 478.091,Z 582.543,A -85,B 0,C 180,E1 -14674.201,E2 -14674.201} C_VEL
LIN {X 0,Y 478.21,Z 582.955,A -85,B 0,C 180,E1 -14675.885,E2 -14675.885} C_VEL
LIN {X 0,Y 478.383,Z 582.083,A -85,B 0,C 180,E1 -14677.572,E2 -14677.572} C_VEL
LIN {X 0,Y 478.642,Z 579.901,A -85,B 0,C 180,E1 -14679.264,E2 -14679.264} C_VEL
LIN {X 0,Y 479.202,Z 576.321,A -85,B 0,C 180,E1 -14680.954,E2 -14680.954} C_VEL
LIN {X 0,Y 479.812,Z 571.256,A -85,B 0,C 180,E1 -14682.649,E2 -14682.649} C_VEL
LIN {X 0,Y 480.465,Z 566.308,A -85,B 0,C 180,E1 -14683.919,E2 -14683.919} C_VEL
LIN {X 0,Y 481.327,Z 559.219,A -85,B 0,C 180,E1 -14685.402,E2 -14685.402} C_VEL
LIN {X 0,Y 482.238,Z 551.447,A -85,B 0,C 180,E1 -14686.721,E2 -14686.721} C_VEL
LIN {X 0,Y 483.203,Z 542.769,A -85,B 0,C 180,E1 -14687.941,E2 -14687.941} C_VEL
LIN {X 0,Y 484.237,Z 531.835,A -85,B 0,C 180,E1 -14689.213,E2 -14689.213} C_VEL
LIN {X 0,Y 485.211,Z 520.617,A -85,B 0,C 180,E1 -14690.271,E2 -14690.271} C_VEL
LIN {X 0,Y 486.201,Z 508.152,A -85,B 0,C 180,E1 -14691.221,E2 -14691.221} C_VEL
LIN {X 0,Y 486.961,Z 496.043,A -85,B 0,C 180,E1 -14691.962,E2 -14691.962} C_VEL
LIN {X 0,Y 487.347,Z 485.246,A -85,B 0,C 180,E1 -14692.499,E2 -14692.499} C_VEL
LIN {X 0,Y 487.792,Z 471.222,A -85,B 0,C 180,E1 -14693.018,E2 -14693.018} C_VEL
LIN {X 0,Y 488.004,Z 458.073,A -85,B 0,C 180,E1 -14693.35,E2 -14693.35} C_VEL
LIN {X 0,Y 489.241,Z 363.329,A -85,B 0,C 180,E1 -14694.776,E2 -14694.776} C_VEL
LIN {X 0,Y 480.605,Z 343.277,A -85,B 0,C 180,E1 -14695.521,E2 -14695.521} C_VEL
LIN {X 0,Y 478.793,Z 338.926,A -85,B 0,C 180,E1 -14695.684,E2 -14695.684} C_VEL
LIN {X 0,Y 478.709,Z 338.416,A -85,B 0,C 180,E1 -14695.728,E2 -14695.728} C_VEL
LIN {X 0,Y 478.745,Z 338.411,A -85,B 0,C 180,E1 -14698.87,E2 -14698.87} C_VEL
LIN {X 0,Y 478.671,Z 338.418,A -85,B 0,C 180,E1 -14701.927,E2 -14701.927} C_VEL
LIN {X 0,Y 478.706,Z 338.412,A -85,B 0,C 180,E1 -14704.975,E2 -14704.975} C_VEL
LIN {X 0,Y 478.673,Z 338.417,A -85,B 0,C 180,E1 -14707.922,E2 -14707.922} C_VEL
LIN {X 0,Y 478.705,Z 338.417,A -85,B 0,C 180,E1 -14710.459,E2 -14710.459} C_VEL
LIN {X 0,Y 478.708,Z 338.413,A -85,B 0,C 180,E1 -14713.449,E2 -14713.449} C_VEL
LIN {X 0,Y 478.744,Z 338.408,A -85,B 0,C 180,E1 -14716.555,E2 -14716.555} C_VEL
LIN {X 0,Y 478.707,Z 338.412,A -85,B 0,C 180,E1 -14719.541,E2 -14719.541} C_VEL
LIN {X 0,Y 478.672,Z 338.393,A -85,B 0,C 180,E1 -14722.203,E2 -14722.203} C_VEL
LIN {X 0,Y 478.722,Z 338.395,A -85,B 0,C 180,E1 -14725.205,E2 -14725.205} C_VEL
LIN {X 0,Y 478.682,Z 338.41,A -85,B 0,C 180,E1 -14728.211,E2 -14728.211} C_VEL
LIN {X 0,Y 478.752,Z 338.404,A -85,B 0,C 180,E1 -14731.383,E2 -14731.383} C_VEL
LIN {X 0,Y 478.742,Z 338.399,A -85,B 0,C 180,E1 -14734.893,E2 -14734.893} C_VEL
LIN {X 0,Y 478.711,Z 338.412,A -85,B 0,C 180,E1 -14737.639,E2 -14737.639} C_VEL
LIN {X 0,Y 478.773,Z 338.407,A -85,B 0,C 180,E1 -14740.592,E2 -14740.592} C_VEL
LIN {X 0,Y 484.214,Z 357.079,A -85,B 0,C 180,E1 -14741.103,E2 -14741.103} C_VEL
LIN {X 0,Y 482.429,Z 456.674,A -85,B 0,C 180,E1 -14742.983,E2 -14742.983} C_VEL
LIN {X 0,Y 482.237,Z 471.763,A -85,B 0,C 180,E1 -14743.437,E2 -14743.437} C_VEL
LIN {X 0,Y 481.856,Z 485.735,A -85,B 0,C 180,E1 -14744.021,E2 -14744.021} C_VEL
LIN {X 0,Y 481.481,Z 498.514,A -85,B 0,C 180,E1 -14744.711,E2 -14744.711} C_VEL
LIN {X 0,Y 481.03,Z 511.107,A -85,B 0,C 180,E1 -14745.56,E2 -14745.56} C_VEL
LIN {X 0,Y 480.409,Z 523.811,A -85,B 0,C 180,E1 -14746.617,E2 -14746.617} C_VEL
LIN {X 0,Y 479.89,Z 535.42,A -85,B 0,C 180,E1 -14747.794,E2 -14747.794} C_VEL
LIN {X 0,Y 479.441,Z 545.643,A -85,B 0,C 180,E1 -14749.051,E2 -14749.051} C_VEL
LIN {X 0,Y 478.987,Z 554.177,A -85,B 0,C 180,E1 -14750.318,E2 -14750.318} C_VEL
LIN {X 0,Y 478.58,Z 562.343,A -85,B 0,C 180,E1 -14751.796,E2 -14751.796} C_VEL
LIN {X 0,Y 478.293,Z 568.913,A -85,B 0,C 180,E1 -14753.272,E2 -14753.272} C_VEL
LIN {X 0,Y 478.15,Z 573.41,A -85,B 0,C 180,E1 -14754.536,E2 -14754.536} C_VEL
LIN {X 0,Y 478.089,Z 576.976,A -85,B 0,C 180,E1 -14755.799,E2 -14755.799} C_VEL
LIN {X 0,Y 478.148,Z 580.34,A -85,B 0,C 180,E1 -14757.481,E2 -14757.481} C_VEL
LIN {X 0,Y 478.12,Z 582.282,A -85,B 0,C 180,E1 -14759.16,E2 -14759.16} C_VEL
LIN {X 0,Y 478.244,Z 582.804,A -85,B 0,C 180,E1 -14760.839,E2 -14760.839} C_VEL
LIN {X 0,Y 478.586,Z 581.842,A -85,B 0,C 180,E1 -14762.516,E2 -14762.516} C_VEL
LIN {X 0,Y 479.225,Z 579.416,A -85,B 0,C 180,E1 -14764.191,E2 -14764.191} C_VEL
LIN {X 0,Y 479.807,Z 575.533,A -85,B 0,C 180,E1 -14765.865,E2 -14765.865} C_VEL
LIN {X 0,Y 480.294,Z 571.797,A -85,B 0,C 180,E1 -14767.048,E2 -14767.048} C_VEL
LIN {X 0,Y 481.189,Z 566.529,A -85,B 0,C 180,E1 -14768.37,E2 -14768.37} C_VEL
LIN {X 0,Y 482.113,Z 559.3,A -85,B 0,C 180,E1 -14769.829,E2 -14769.829} C_VEL
LIN {X 0,Y 483.029,Z 551.682,A -85,B 0,C 180,E1 -14771.077,E2 -14771.077} C_VEL
LIN {X 0,Y 484.048,Z 542.527,A -85,B 0,C 180,E1 -14772.324,E2 -14772.324} C_VEL
LIN {X 0,Y 484.994,Z 532.403,A -85,B 0,C 180,E1 -14773.467,E2 -14773.467} C_VEL
LIN {X 0,Y 486.106,Z 521.134,A -85,B 0,C 180,E1 -14774.499,E2 -14774.499} C_VEL
LIN {X 0,Y 487.217,Z 508.318,A -85,B 0,C 180,E1 -14775.458,E2 -14775.458} C_VEL
LIN {X 0,Y 488.057,Z 495.137,A -85,B 0,C 180,E1 -14776.252,E2 -14776.252} C_VEL
LIN {X 0,Y 488.587,Z 481.224,A -85,B 0,C 180,E1 -14776.903,E2 -14776.903} C_VEL
LIN {X 0,Y 489.06,Z 465.912,A -85,B 0,C 180,E1 -14777.423,E2 -14777.423} C_VEL
LIN {X 0,Y 489.869,Z 436.976,A -85,B 0,C 180,E1 -14778.065,E2 -14778.065} C_VEL
LIN {X 0,Y 492.91,Z 366.215,A -85,B 0,C 180,E1 -14779.602,E2 -14779.602} C_VEL
LIN {X 0,Y 486.619,Z 353.3,A -85,B 0,C 180,E1 -14780.441,E2 -14780.441} C_VEL
LIN {X 0,Y 482,Z 344.906,A -85,B 0,C 180,E1 -14781.074,E2 -14781.074} C_VEL
LIN {X 0,Y 480.208,Z 341.865,A -85,B 0,C 180,E1 -14781.323,E2 -14781.323} C_VEL
LIN {X 0,Y 478.889,Z 339.174,A -85,B 0,C 180,E1 -14781.522,E2 -14781.522} C_VEL
LIN {X 0,Y 478.751,Z 338.41,A -85,B 0,C 180,E1 -14781.567,E2 -14781.567} C_VEL
LIN {X 0,Y 478.749,Z 338.409,A -85,B 0,C 180,E1 -14784.891,E2 -14784.891} C_VEL
LIN {X 0,Y 478.765,Z 338.408,A -85,B 0,C 180,E1 -14787.915,E2 -14787.915} C_VEL
LIN {X 0,Y 478.723,Z 338.41,A -85,B 0,C 180,E1 -14790.804,E2 -14790.804} C_VEL
LIN {X 0,Y 478.757,Z 338.403,A -85,B 0,C 180,E1 -14793.777,E2 -14793.777} C_VEL
LIN {X 0,Y 478.742,Z 338.402,A -85,B 0,C 180,E1 -14796.86,E2 -14796.86} C_VEL
LIN {X 0,Y 478.723,Z 338.403,A -85,B 0,C 180,E1 -14800.075,E2 -14800.075} C_VEL
LIN {X 0,Y 478.742,Z 338.406,A -85,B 0,C 180,E1 -14803.445,E2 -14803.445} C_VEL
LIN {X 0,Y 478.741,Z 338.406,A -85,B 0,C 180,E1 -14806.555,E2 -14806.555} C_VEL
LIN {X 0,Y 478.704,Z 338.411,A -85,B 0,C 180,E1 -14809.541,E2 -14809.541} C_VEL
LIN {X 0,Y 478.67,Z 338.417,A -85,B 0,C 180,E1 -14812.203,E2 -14812.203} C_VEL
LIN {X 0,Y 478.694,Z 338.406,A -85,B 0,C 180,E1 -14815.203,E2 -14815.203} C_VEL
LIN {X 0,Y 478.726,Z 338.536,A -85,B 0,C 180,E1 -14817.851,E2 -14817.851} C_VEL
LIN {X 0,Y 482.817,Z 355.305,A -85,B 0,C 180,E1 -14820.511,E2 -14820.511} C_VEL
LIN {X 0,Y 485.21,Z 367.259,A -85,B 0,C 180,E1 -14822.316,E2 -14822.316} C_VEL
LIN {X 0,Y 483.87,Z 383.471,A -85,B 0,C 180,E1 -14824.49,E2 -14824.49} C_VEL
LIN {X 0,Y 482.077,Z 406.715,A -85,B 0,C 180,E1 -14827.579,E2 -14827.579} C_VEL
LIN {X 0,Y 481.861,Z 410.068,A -85,B 0,C 180,E1 -14828.022,E2 -14828.022} C_VEL
LIN {X 0,Y 486.245,Z 439.352,A -85,B 0,C 180,E1 -14829.128,E2 -14829.128} C_VEL
LIN {X 0,Y 488.608,Z 468.058,A -85,B 0,C 180,E1 -14830.013,E2 -14830.013} C_VEL
LIN {X 0,Y 488.69,Z 474.1,A -85,B 0,C 180,E1 -14830.167,E2 -14830.167} C_VEL
LIN {X 0,Y 487.009,Z 517.729,A -85,B 0,C 180,E1 -14831.091,E2 -14831.091} C_VEL
LIN {X 0,Y 486.304,Z 560.299,A -85,B 0,C 180,E1 -14831.743,E2 -14831.743} C_VEL
LIN {X 0,Y 485.567,Z 574.691,A -85,B 0,C 180,E1 -14832.122,E2 -14832.122} C_VEL
LIN {X 0,Y 484.493,Z 588.89,A -85,B 0,C 180,E1 -14832.668,E2 -14832.668} C_VEL
LIN {X 0,Y 483.359,Z 602.386,A -85,B 0,C 180,E1 -14833.369,E2 -14833.369} C_VEL
LIN {X 0,Y 482.185,Z 614.815,A -85,B 0,C 180,E1 -14834.194,E2 -14834.194} C_VEL
LIN {X 0,Y 480.894,Z 627.388,A -85,B 0,C 180,E1 -14835.232,E2 -14835.232} C_VEL
LIN {X 0,Y 479.848,Z 637.715,A -85,B 0,C 180,E1 -14836.278,E2 -14836.278} C_VEL
LIN {X 0,Y 479.194,Z 645.642,A -85,B 0,C 180,E1 -14837.227,E2 -14837.227} C_VEL
LIN {X 0,Y 478.548,Z 657.863,A -85,B 0,C 180,E1 -14838.411,E2 -14838.411} C_VEL
LIN {X 0,Y 478.063,Z 668.419,A -85,B 0,C 180,E1 -14839.66,E2 -14839.66} C_VEL
LIN {X 0,Y 477.626,Z 677.245,A -85,B 0,C 180,E1 -14840.929,E2 -14840.929} C_VEL
LIN {X 0,Y 477.277,Z 685.612,A -85,B 0,C 180,E1 -14842.41,E2 -14842.41} C_VEL
LIN {X 0,Y 477.146,Z 691.463,A -85,B 0,C 180,E1 -14843.679,E2 -14843.679} C_VEL
LIN {X 0,Y 477.033,Z 696.207,A -85,B 0,C 180,E1 -14844.946,E2 -14844.946} C_VEL
LIN {X 0,Y 476.951,Z 699.908,A -85,B 0,C 180,E1 -14846.211,E2 -14846.211} C_VEL
LIN {X 0,Y 476.942,Z 702.711,A -85,B 0,C 180,E1 -14847.475,E2 -14847.475} C_VEL
LIN {X 0,Y 476.942,Z 705.099,A -85,B 0,C 180,E1 -14849.158,E2 -14849.158} C_VEL
LIN {X 0,Y 476.923,Z 706.007,A -85,B 0,C 180,E1 -14850.841,E2 -14850.841} C_VEL
LIN {X 0,Y 476.942,Z 705.444,A -85,B 0,C 180,E1 -14852.525,E2 -14852.525} C_VEL
LIN {X 0,Y 477.01,Z 703.393,A -85,B 0,C 180,E1 -14854.21,E2 -14854.21} C_VEL
LIN {X 0,Y 477.282,Z 699.819,A -85,B 0,C 180,E1 -14855.896,E2 -14855.896} C_VEL
LIN {X 0,Y 477.622,Z 694.653,A -85,B 0,C 180,E1 -14857.584,E2 -14857.584} C_VEL
LIN {X 0,Y 478.088,Z 689.644,A -85,B 0,C 180,E1 -14858.849,E2 -14858.849} C_VEL
LIN {X 0,Y 478.845,Z 682.397,A -85,B 0,C 180,E1 -14860.323,E2 -14860.323} C_VEL
LIN {X 0,Y 479.731,Z 673.428,A -85,B 0,C 180,E1 -14861.795,E2 -14861.795} C_VEL
LIN {X 0,Y 480.675,Z 664.07,A -85,B 0,C 180,E1 -14863.054,E2 -14863.054} C_VEL
LIN {X 0,Y 481.913,Z 652.641,A -85,B 0,C 180,E1 -14864.305,E2 -14864.305} C_VEL
LIN {X 0,Y 482.94,Z 641.147,A -85,B 0,C 180,E1 -14865.349,E2 -14865.349} C_VEL
LIN {X 0,Y 484.178,Z 628.54,A -85,B 0,C 180,E1 -14866.278,E2 -14866.278} C_VEL
LIN {X 0,Y 485.304,Z 614.55,A -85,B 0,C 180,E1 -14867.102,E2 -14867.102} C_VEL
LIN {X 0,Y 486.351,Z 599.861,A -85,B 0,C 180,E1 -14867.759,E2 -14867.759} C_VEL
LIN {X 0,Y 487.257,Z 585.012,A -85,B 0,C 180,E1 -14868.24,E2 -14868.24} C_VEL
LIN {X 0,Y 491.653,Z 483.546,A -85,B 0,C 180,E1 -14870.474,E2 -14870.474} C_VEL
LIN {X 0,Y 492.074,Z 471.92,A -85,B 0,C 180,E1 -14870.75,E2 -14870.75} C_VEL
LIN {X 0,Y 491,Z 453.928,A -85,B 0,C 180,E1 -14871.312,E2 -14871.312} C_VEL
LIN {X 0,Y 488.897,Z 435.636,A -85,B 0,C 180,E1 -14872.002,E2 -14872.002} C_VEL
LIN {X 0,Y 487.864,Z 419.234,A -85,B 0,C 180,E1 -14872.963,E2 -14872.963} C_VEL
LIN {X 0,Y 486.295,Z 397.464,A -85,B 0,C 180,E1 -14874.42,E2 -14874.42} C_VEL
LIN {X 0,Y 485.166,Z 382.726,A -85,B 0,C 180,E1 -14875.551,E2 -14875.551} C_VEL
LIN {X 0,Y 484.401,Z 371.468,A -85,B 0,C 180,E1 -14876.491,E2 -14876.491} C_VEL
LIN {X 0,Y 483.731,Z 362.111,A -85,B 0,C 180,E1 -14877.37,E2 -14877.37} C_VEL
LIN {X 0,Y 482.02,Z 353.825,A -85,B 0,C 180,E1 -14878.418,E2 -14878.418} C_VEL
LIN {X 0,Y 478.749,Z 338.406,A -85,B 0,C 180,E1 -14880.704,E2 -14880.704} C_VEL
LIN {X 0,Y 478.654,Z 338.417,A -85,B 0,C 180,E1 -14883.785,E2 -14883.785} C_VEL
LIN {X 0,Y 478.665,Z 338.419,A -85,B 0,C 180,E1 -14886.867,E2 -14886.867} C_VEL
LIN {X 0,Y 478.688,Z 338.413,A -85,B 0,C 180,E1 -14890.078,E2 -14890.078} C_VEL
LIN {X 0,Y 478.706,Z 338.415,A -85,B 0,C 180,E1 -14892.979,E2 -14892.979} C_VEL
LIN {X 0,Y 478.727,Z 338.412,A -85,B 0,C 180,E1 -14895.802,E2 -14895.802} C_VEL
LIN {X 0,Y 478.705,Z 338.411,A -85,B 0,C 180,E1 -14898.819,E2 -14898.819} C_VEL
LIN {X 0,Y 478.699,Z 338.475,A -85,B 0,C 180,E1 -14901.948,E2 -14901.948} C_VEL
LIN {X 0,Y 483.138,Z 348.466,A -85,B 0,C 180,E1 -14904.556,E2 -14904.556} C_VEL
LIN {X 0,Y 486.422,Z 356.8,A -85,B 0,C 180,E1 -14906.396,E2 -14906.396} C_VEL
LIN {X 0,Y 489.774,Z 367.202,A -85,B 0,C 180,E1 -14908.403,E2 -14908.403} C_VEL
LIN {X 0,Y 492.274,Z 377.181,A -85,B 0,C 180,E1 -14910.132,E2 -14910.132} C_VEL
LIN {X 0,Y 493.083,Z 382.764,A -85,B 0,C 180,E1 -14910.982,E2 -14910.982} C_VEL
LIN {X 0,Y 490.421,Z 409.146,A -85,B 0,C 180,E1 -14914.234,E2 -14914.234} C_VEL
LIN {X 0,Y 487.91,Z 437.177,A -85,B 0,C 180,E1 -14917.64,E2 -14917.64} C_VEL
LIN {X 0,Y 487.73,Z 439.937,A -85,B 0,C 180,E1 -14917.95,E2 -14917.95} C_VEL
LIN {X 0,Y 491.302,Z 459.028,A -85,B 0,C 180,E1 -14918.756,E2 -14918.756} C_VEL
LIN {X 0,Y 492.695,Z 470.621,A -85,B 0,C 180,E1 -14919.165,E2 -14919.165} C_VEL
LIN {X 0,Y 488.945,Z 555.755,A -85,B 0,C 180,E1 -14921.031,E2 -14921.031} C_VEL
LIN {X 0,Y 487.802,Z 583.247,A -85,B 0,C 180,E1 -14921.639,E2 -14921.639} C_VEL
LIN {X 0,Y 486.886,Z 596.934,A -85,B 0,C 180,E1 -14922.091,E2 -14922.091} C_VEL
LIN {X 0,Y 485.852,Z 610.577,A -85,B 0,C 180,E1 -14922.702,E2 -14922.702} C_VEL
LIN {X 0,Y 484.748,Z 624.795,A -85,B 0,C 180,E1 -14923.527,E2 -14923.527} C_VEL
LIN {X 0,Y 483.533,Z 637.581,A -85,B 0,C 180,E1 -14924.455,E2 -14924.455} C_VEL
LIN {X 0,Y 482.301,Z 649.195,A -85,B 0,C 180,E1 -14925.492,E2 -14925.492} C_VEL
LIN {X 0,Y 481.288,Z 658.965,A -85,B 0,C 180,E1 -14926.535,E2 -14926.535} C_VEL
LIN {X 0,Y 480.177,Z 668.721,A -85,B 0,C 180,E1 -14927.781,E2 -14927.781} C_VEL
LIN {X 0,Y 479.313,Z 678.185,A -85,B 0,C 180,E1 -14929.262,E2 -14929.262} C_VEL
LIN {X 0,Y 478.353,Z 685.84,A -85,B 0,C 180,E1 -14930.731,E2 -14930.731} C_VEL
LIN {X 0,Y 477.859,Z 691.117,A -85,B 0,C 180,E1 -14931.996,E2 -14931.996} C_VEL
LIN {X 0,Y 477.372,Z 696.669,A -85,B 0,C 180,E1 -14933.682,E2 -14933.682} C_VEL
LIN {X 0,Y 477.098,Z 699.729,A -85,B 0,C 180,E1 -14934.947,E2 -14934.947} C_VEL
LIN {X 0,Y 476.942,Z 702.524,A -85,B 0,C 180,E1 -14936.632,E2 -14936.632} C_VEL
LIN {X 0,Y 476.851,Z 703.837,A -85,B 0,C 180,E1 -14938.317,E2 -14938.317} C_VEL
LIN {X 0,Y 476.853,Z 703.685,A -85,B 0,C 180,E1 -14940,E2 -14940} C_VEL
LIN {X 0,Y 476.847,Z 702.081,A -85,B 0,C 180,E1 -14941.684,E2 -14941.684} C_VEL
LIN {X 0,Y 476.889,Z 699,A -85,B 0,C 180,E1 -14943.368,E2 -14943.368} C_VEL
LIN {X 0,Y 476.98,Z 694.358,A -85,B 0,C 180,E1 -14945.055,E2 -14945.055} C_VEL
LIN {X 0,Y 477.117,Z 689.706,A -85,B 0,C 180,E1 -14946.322,E2 -14946.322} C_VEL
LIN {X 0,Y 477.384,Z 682.956,A -85,B 0,C 180,E1 -14947.801,E2 -14947.801} C_VEL
LIN {X 0,Y 477.79,Z 674.489,A -85,B 0,C 180,E1 -14949.28,E2 -14949.28} C_VEL
LIN {X 0,Y 478.274,Z 665.622,A -85,B 0,C 180,E1 -14950.549,E2 -14950.549} C_VEL
LIN {X 0,Y 478.817,Z 654.886,A -85,B 0,C 180,E1 -14951.818,E2 -14951.818} C_VEL
LIN {X 0,Y 479.46,Z 642.927,A -85,B 0,C 180,E1 -14952.98,E2 -14952.98} C_VEL
LIN {X 0,Y 480.076,Z 630.943,A -85,B 0,C 180,E1 -14953.93,E2 -14953.93} C_VEL
LIN {X 0,Y 480.819,Z 617.822,A -85,B 0,C 180,E1 -14954.77,E2 -14954.77} C_VEL
LIN {X 0,Y 481.355,Z 604.305,A -85,B 0,C 180,E1 -14955.455,E2 -14955.455} C_VEL
LIN {X 0,Y 481.845,Z 589.882,A -85,B 0,C 180,E1 -14956.007,E2 -14956.007} C_VEL
LIN {X 0,Y 482.3,Z 575.199,A -85,B 0,C 180,E1 -14956.391,E2 -14956.391} C_VEL
LIN {X 0,Y 484.471,Z 466.199,A -85,B 0,C 180,E1 -14958.47,E2 -14958.47} C_VEL
LIN {X 0,Y 481.662,Z 439.626,A -85,B 0,C 180,E1 -14959.074,E2 -14959.074} C_VEL
LIN {X 0,Y 483.085,Z 409.423,A -85,B 0,C 180,E1 -14962.597,E2 -14962.597} C_VEL
LIN {X 0,Y 484.408,Z 384.765,A -85,B 0,C 180,E1 -14965.479,E2 -14965.479} C_VEL
